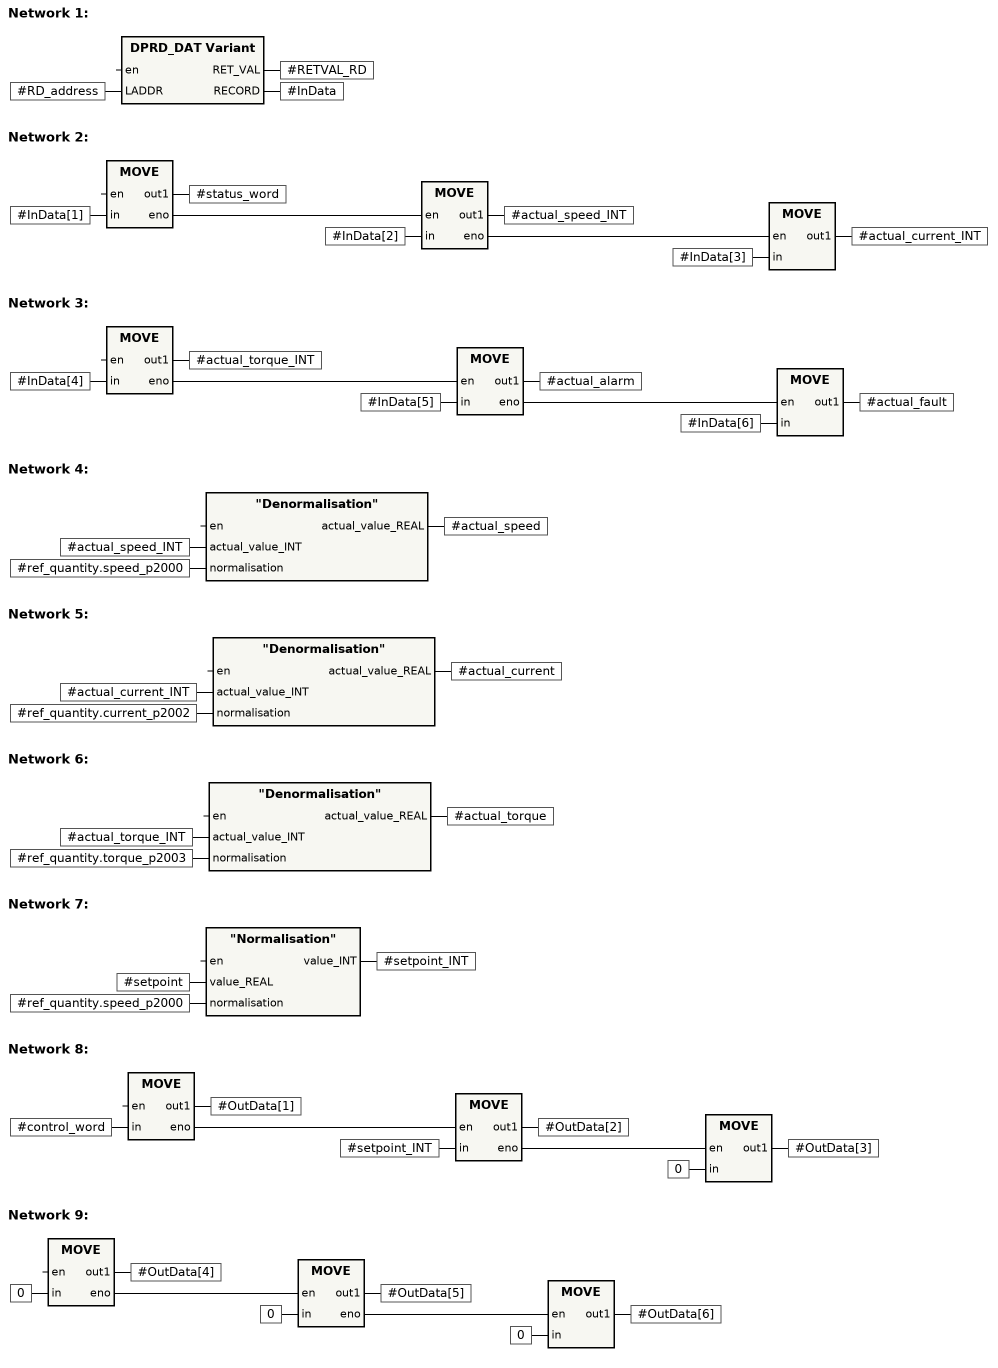
   #RETVAL_RD := DPRD_DAT(LADDR := #RD_address, RECORD => #InData);
END_REGION

REGION Network 2
   // ENO of a box is taken as its EN; it also drops when the box reports an error
   #status_word := #InData[1];
   #actual_speed_INT := #InData[2];
   #actual_current_INT := #InData[3];
END_REGION

REGION Network 3
   // ENO of a box is taken as its EN; it also drops when the box reports an error
   #actual_torque_INT := #InData[4];
   #actual_alarm := #InData[5];
   #actual_fault := #InData[6];
END_REGION

REGION Network 4
   "Denormalisation"(actual_value_INT := #actual_speed_INT,
                     normalisation := #ref_quantity.speed_p2000,
                     actual_value_REAL => #actual_speed);
END_REGION

REGION Network 5
   "Denormalisation"(actual_value_INT := #actual_current_INT,
                     normalisation := #ref_quantity.current_p2002,
                     actual_value_REAL => #actual_current);
END_REGION

REGION Network 6
   "Denormalisation"(actual_value_INT := #actual_torque_INT,
                     normalisation := #ref_quantity.torque_p2003,
                     actual_value_REAL => #actual_torque);
END_REGION

REGION Network 7
   "Normalisation"(value_REAL := #setpoint,
                   normalisation := #ref_quantity.speed_p2000,
                   value_INT => #setpoint_INT);
END_REGION

REGION Network 8
   // ENO of a box is taken as its EN; it also drops when the box reports an error
   #OutData[1] := #control_word;
   #OutData[2] := #setpoint_INT;
   #OutData[3] := 0;
END_REGION

REGION Network 9
   // ENO of a box is taken as its EN; it also drops when the box reports an error
   #OutData[4] := 0;
   #OutData[5] := 0;
   #OutData[6] := 0;
END_REGION

REGION Network 10
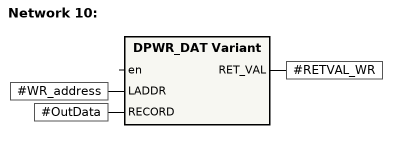
   #RETVAL_WR := DPWR_DAT(LADDR := #WR_address, RECORD := #OutData);
END_REGION
END_FUNCTION_BLOCK

FUNCTION "Denormalisation" : Void   // FC14, FBD
{ S7_Optimized_Access := 'TRUE' }
VERSION : 0.1
// stored: AutoNumber true, IsIECCheckEnabled false, SetENOAutomatically false, UDAEnableTagReadback false
   VAR_INPUT
      actual_value_INT : Int;
      normalisation : Real;
   END_VAR
   VAR_OUTPUT
      actual_value_REAL : Real;
   END_VAR
   VAR_TEMP
      temp_actual_value_DINT : DInt;
      temp_actual_value_REAL : Real;
   END_VAR
BEGIN

REGION Network 1
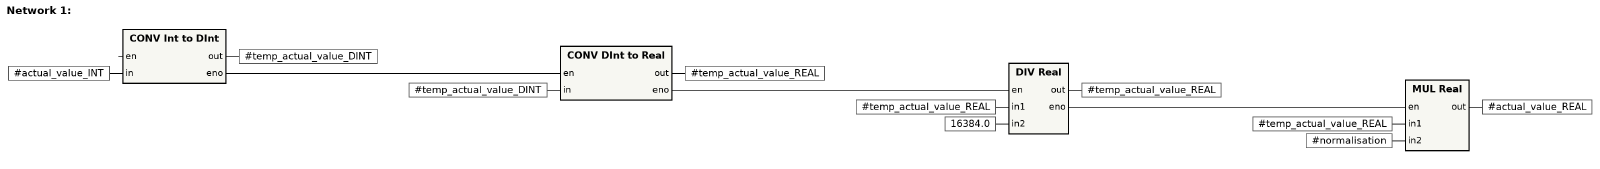
   // ENO of a box is taken as its EN; it also drops when the box reports an error
   #temp_actual_value_DINT := INT_TO_DINT(#actual_value_INT);
   #temp_actual_value_REAL := DINT_TO_REAL(#temp_actual_value_DINT);
   #temp_actual_value_REAL := #temp_actual_value_REAL / 16384.0;
   #actual_value_REAL := #temp_actual_value_REAL * #normalisation;
END_REGION
END_FUNCTION

FUNCTION "Normalisation" : Void   // FC15, FBD
{ S7_Optimized_Access := 'TRUE' }
VERSION : 0.1
// stored: AutoNumber true, IsIECCheckEnabled false, SetENOAutomatically false, UDAEnableTagReadback false
   VAR_INPUT
      value_REAL : Real;
      normalisation : Real;
   END_VAR
   VAR_OUTPUT
      value_INT : Int;
   END_VAR
   VAR_TEMP
      temp_value_DINT : DInt;
      temp_value_REAL : Real;
   END_VAR
BEGIN

REGION Network 1
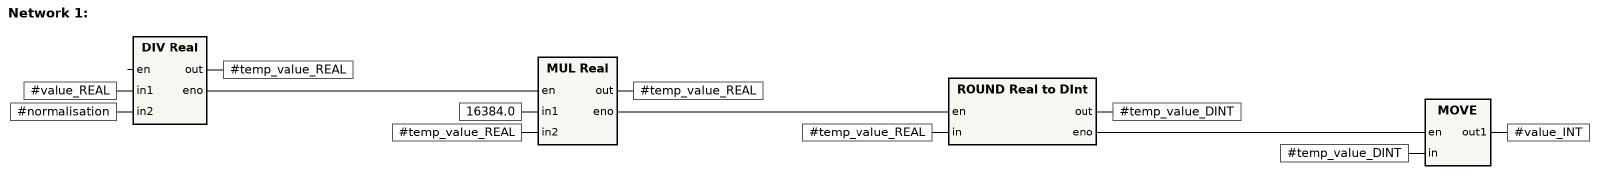
   // ENO of a box is taken as its EN; it also drops when the box reports an error
   #temp_value_REAL := #value_REAL / #normalisation;
   #temp_value_REAL := 16384.0 * #temp_value_REAL;
   #temp_value_DINT := ROUND(#temp_value_REAL);
   #value_INT := #temp_value_DINT;
END_REGION
END_FUNCTION

FUNCTION "FC09_NoPressurePlate" : Void   // FC9, LAD
TITLE = Pressure palte isn't present
{ S7_Optimized_Access := 'FALSE' }
AUTHOR : Robopac
VERSION : 0.0
// stored: AutoNumber false, IsIECCheckEnabled false, SetENOAutomatically false, UDAEnableTagReadback false
BEGIN

REGION Network 1: Pressure plate bits
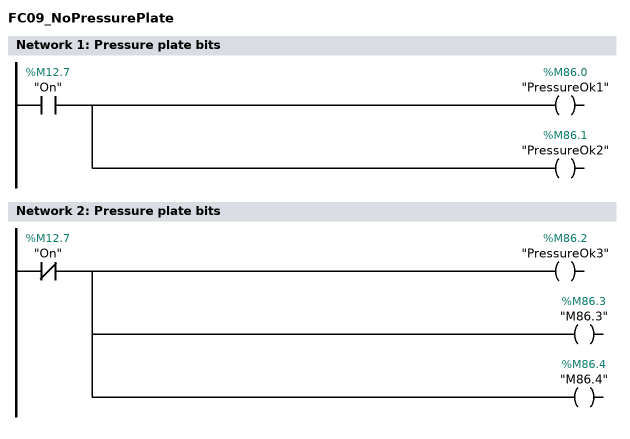
   RUNG wire#powerrail
      Contact( "On" )
      wire#w1
      Coil( "PressureOk1" )
   END_RUNG
   RUNG wire#w1
      Coil( "PressureOk2" )
   END_RUNG
   // the same network as SCL:
   "PressureOk1" := "On";
   "PressureOk2" := "On";
END_REGION

REGION Network 2: Pressure plate bits
   RUNG wire#powerrail
      I_Contact( "On" )
      wire#w1
      Coil( "PressureOk3" )
   END_RUNG
   RUNG wire#w1
      Coil( "M86.3" )
   END_RUNG
   RUNG wire#w1
      Coil( "M86.4" )
   END_RUNG
   // the same network as SCL:
   "PressureOk3" := NOT "On";
   "M86.3" := NOT "On";
   "M86.4" := NOT "On";
END_REGION
END_FUNCTION

FUNCTION "FC11_PressureRectangularPn5W" : Void   // FC11, LAD
{ S7_Optimized_Access := 'FALSE' }
VERSION : 0.1
// stored: AutoNumber false, IsIECCheckEnabled false, SetENOAutomatically false, UDAEnableTagReadback false
BEGIN

REGION Network 1: Timeout for pressure plate upward/downward
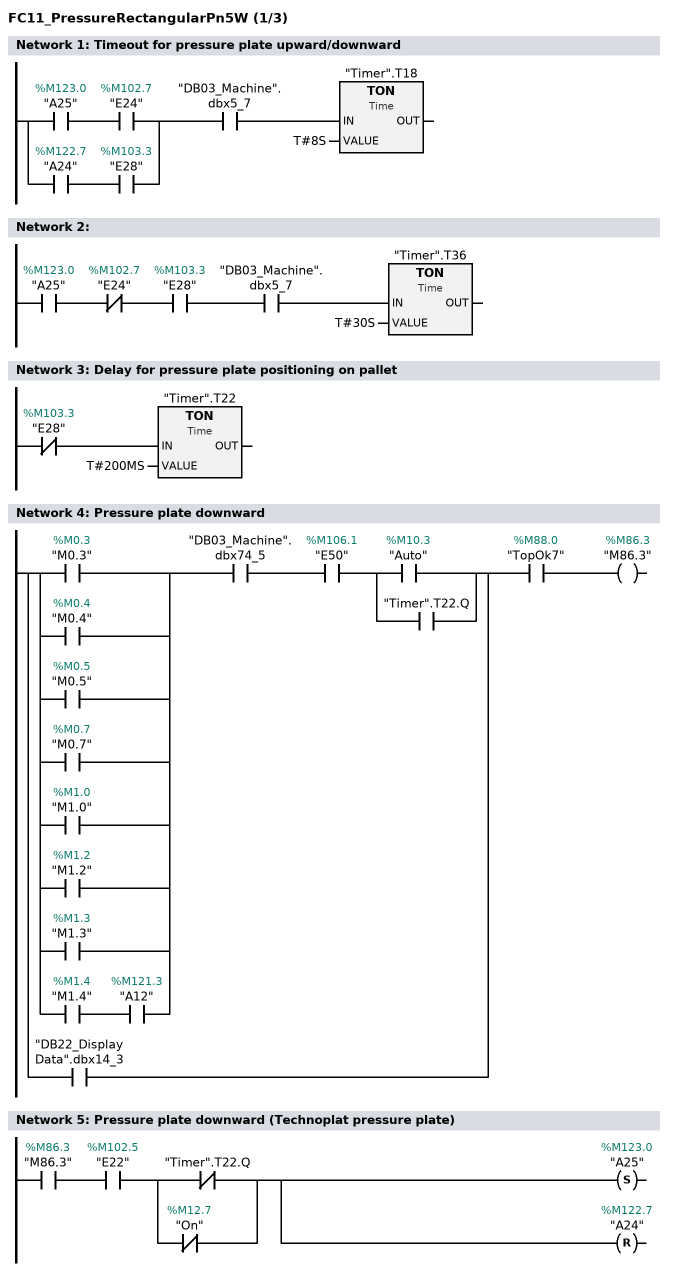
   "Timer".T18.TON(IN := (("A25" AND "E24") OR ("A24" AND "E28")) AND "DB03_Machine".dbx5_7, PT := T#8S);   // TON coil
END_REGION

REGION Network 2
   "Timer".T36.TON(IN := "A25" AND NOT "E24" AND "E28" AND "DB03_Machine".dbx5_7, PT := T#30S);   // TON coil
END_REGION

REGION Network 3: Delay for pressure plate positioning on pallet
   "Timer".T22.TON(IN := NOT "E28", PT := T#200MS);   // TON coil
END_REGION

REGION Network 4: Pressure plate downward
   RUNG wire#powerrail
      Contact( "M0.3" )
      wire#w1
      Contact( "DB03_Machine".dbx74_5 )
      Contact( "E50" )
      wire#w2
      Contact( "Auto" )
      wire#w3
      Contact( "TopOk7" )
      Coil( "M86.3" )
   END_RUNG
   RUNG wire#powerrail
      Contact( "M0.4" )
   END_RUNG wire#w1
   RUNG wire#powerrail
      Contact( "M0.5" )
   END_RUNG wire#w1
   RUNG wire#powerrail
      Contact( "M0.7" )
   END_RUNG wire#w1
   RUNG wire#powerrail
      Contact( "M1.0" )
   END_RUNG wire#w1
   RUNG wire#powerrail
      Contact( "M1.2" )
   END_RUNG wire#w1
   RUNG wire#powerrail
      Contact( "M1.3" )
   END_RUNG wire#w1
   RUNG wire#powerrail
      Contact( "M1.4" )
      Contact( "A12" )
   END_RUNG wire#w1
   RUNG wire#w2
      Contact( "Timer".T22.Q )
   END_RUNG wire#w3
   RUNG wire#powerrail
      Contact( "DB22_DisplayData".dbx14_3 )
   END_RUNG wire#w3
   // the same network as SCL:
   "M86.3" := ((("M0.3" OR "M0.4" OR "M0.5" OR "M0.7" OR "M1.0" OR "M1.2" OR "M1.3" OR ("M1.4" AND "A12")) AND "DB03_Machine".dbx74_5 AND "E50" AND ("Auto" OR "Timer".T22.Q)) OR "DB22_DisplayData".dbx14_3) AND "TopOk7";
END_REGION

REGION Network 5: Pressure plate downward (Technoplat pressure plate)
   RUNG wire#powerrail
      Contact( "M86.3" )
      Contact( "E22" )
      wire#w1
      I_Contact( "Timer".T22.Q )
      wire#w2
      S_Coil( "A25" )
   END_RUNG
   RUNG wire#w1
      I_Contact( "On" )
   END_RUNG wire#w2
   RUNG wire#w2
      R_Coil( "A24" )
   END_RUNG
   // the same network as SCL:
   IF "M86.3" AND "E22" AND (NOT "Timer".T22.Q OR NOT "On") THEN
       "A25" := TRUE;
       "A24" := FALSE;
   END_IF;
END_REGION

REGION Network 6: Pressure plate upward
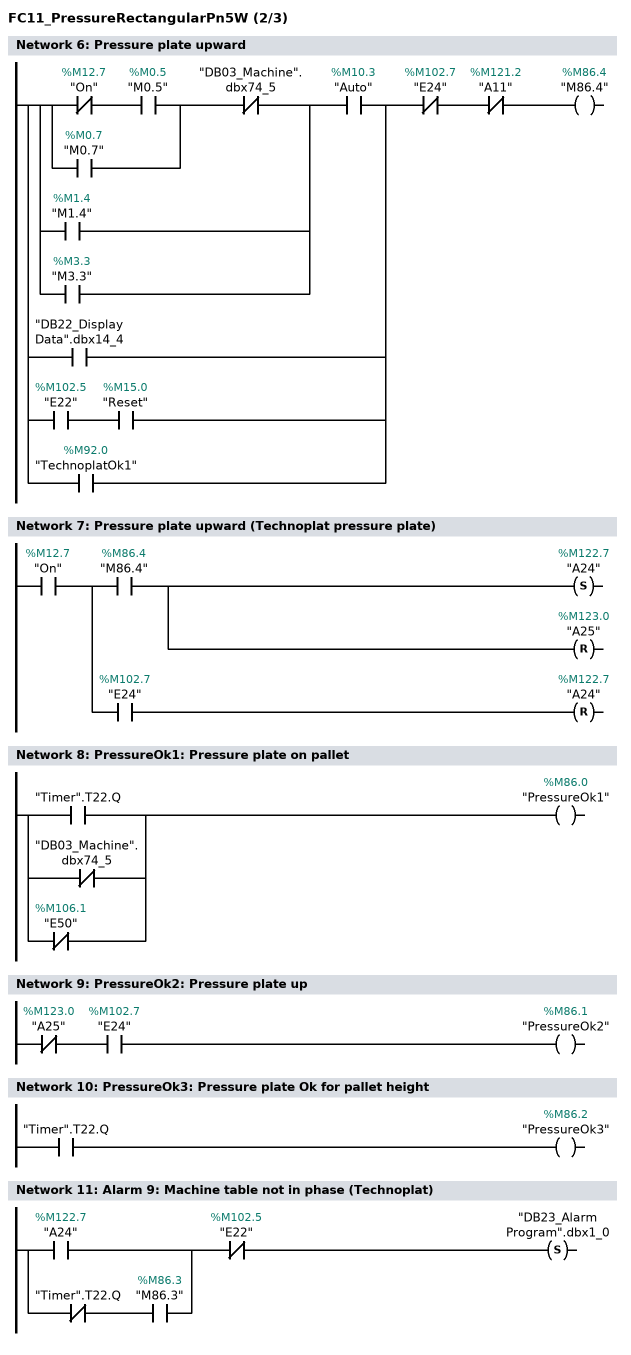
   RUNG wire#powerrail
      I_Contact( "On" )
      Contact( "M0.5" )
      wire#w1
      I_Contact( "DB03_Machine".dbx74_5 )
      wire#w2
      Contact( "Auto" )
      wire#w3
      I_Contact( "E24" )
      I_Contact( "A11" )
      Coil( "M86.4" )
   END_RUNG
   RUNG wire#powerrail
      Contact( "M0.7" )
   END_RUNG wire#w1
   RUNG wire#powerrail
      Contact( "M1.4" )
   END_RUNG wire#w2
   RUNG wire#powerrail
      Contact( "M3.3" )
   END_RUNG wire#w2
   RUNG wire#powerrail
      Contact( "DB22_DisplayData".dbx14_4 )
   END_RUNG wire#w3
   RUNG wire#powerrail
      Contact( "E22" )
      Contact( "Reset" )
   END_RUNG wire#w3
   RUNG wire#powerrail
      Contact( "TechnoplatOk1" )
   END_RUNG wire#w3
   // the same network as SCL:
   "M86.4" := ((((((NOT "On" AND "M0.5") OR "M0.7") AND NOT "DB03_Machine".dbx74_5) OR "M1.4" OR "M3.3") AND "Auto") OR "DB22_DisplayData".dbx14_4 OR ("E22" AND "Reset") OR "TechnoplatOk1") AND NOT "E24" AND NOT "A11";
END_REGION

REGION Network 7: Pressure plate upward (Technoplat pressure plate)
   RUNG wire#powerrail
      Contact( "On" )
      wire#w1
      Contact( "M86.4" )
      wire#w2
      S_Coil( "A24" )
   END_RUNG
   RUNG wire#w2
      R_Coil( "A25" )
   END_RUNG
   RUNG wire#w1
      Contact( "E24" )
      R_Coil( "A24" )
   END_RUNG
   // the same network as SCL:
   IF "On" AND "M86.4" THEN
       "A24" := TRUE;
       "A25" := FALSE;
   END_IF;
   IF "On" AND "E24" THEN "A24" := FALSE; END_IF;
END_REGION

REGION Network 8: PressureOk1: Pressure plate on pallet
   RUNG wire#powerrail
      Contact( "Timer".T22.Q )
      wire#w1
      Coil( "PressureOk1" )
   END_RUNG
   RUNG wire#powerrail
      I_Contact( "DB03_Machine".dbx74_5 )
   END_RUNG wire#w1
   RUNG wire#powerrail
      I_Contact( "E50" )
   END_RUNG wire#w1
   // the same network as SCL:
   "PressureOk1" := "Timer".T22.Q OR NOT "DB03_Machine".dbx74_5 OR NOT "E50";
END_REGION

REGION Network 9: PressureOk2: Pressure plate up
   RUNG wire#powerrail
      I_Contact( "A25" )
      Contact( "E24" )
      Coil( "PressureOk2" )
   END_RUNG
   // the same network as SCL:
   "PressureOk2" := NOT "A25" AND "E24";
END_REGION

REGION Network 10: PressureOk3: Pressure plate Ok for pallet height
   RUNG wire#powerrail
      Contact( "Timer".T22.Q )
      Coil( "PressureOk3" )
   END_RUNG
   // the same network as SCL:
   "PressureOk3" := "Timer".T22.Q;
END_REGION

REGION Network 11: Alarm 9: Machine table not in phase (Technoplat)
   RUNG wire#powerrail
      Contact( "A24" )
      wire#w1
      I_Contact( "E22" )
      S_Coil( "DB23_AlarmProgram".dbx1_0 )
   END_RUNG
   RUNG wire#powerrail
      I_Contact( "Timer".T22.Q )
      Contact( "M86.3" )
   END_RUNG wire#w1
   // the same network as SCL:
   IF ("A24" OR (NOT "Timer".T22.Q AND "M86.3")) AND NOT "E22" THEN
       "DB23_AlarmProgram".dbx1_0 := TRUE;
   END_IF;
END_REGION

REGION Network 12: Alarm 15: Pressure plate not up (Pressure plate)
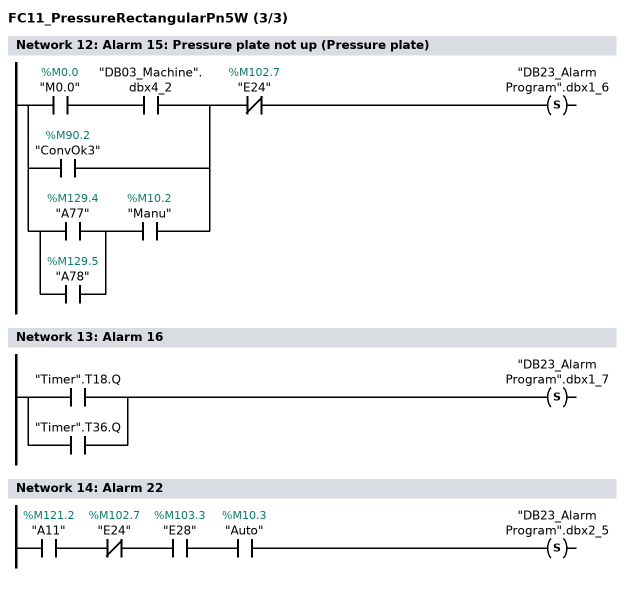
   RUNG wire#powerrail
      Contact( "M0.0" )
      Contact( "DB03_Machine".dbx4_2 )
      wire#w1
      I_Contact( "E24" )
      S_Coil( "DB23_AlarmProgram".dbx1_6 )
   END_RUNG
   RUNG wire#powerrail
      Contact( "ConvOk3" )
   END_RUNG wire#w1
   RUNG wire#powerrail
      Contact( "A77" )
      wire#w2
      Contact( "Manu" )
   END_RUNG wire#w1
   RUNG wire#powerrail
      Contact( "A78" )
   END_RUNG wire#w2
   // the same network as SCL:
   IF (("M0.0" AND "DB03_Machine".dbx4_2) OR "ConvOk3" OR (("A77" OR "A78") AND "Manu")) AND NOT "E24" THEN
       "DB23_AlarmProgram".dbx1_6 := TRUE;
   END_IF;
END_REGION

REGION Network 13: Alarm 16
   RUNG wire#powerrail
      Contact( "Timer".T18.Q )
      wire#w1
      S_Coil( "DB23_AlarmProgram".dbx1_7 )
   END_RUNG
   RUNG wire#powerrail
      Contact( "Timer".T36.Q )
   END_RUNG wire#w1
   // the same network as SCL:
   IF "Timer".T18.Q OR "Timer".T36.Q THEN "DB23_AlarmProgram".dbx1_7 := TRUE; END_IF;
END_REGION

REGION Network 14: Alarm 22
   RUNG wire#powerrail
      Contact( "A11" )
      I_Contact( "E24" )
      Contact( "E28" )
      Contact( "Auto" )
      S_Coil( "DB23_AlarmProgram".dbx2_5 )
   END_RUNG
   // the same network as SCL:
   IF "A11" AND NOT "E24" AND "E28" AND "Auto" THEN "DB23_AlarmProgram".dbx2_5 := TRUE; END_IF;
END_REGION
END_FUNCTION

FUNCTION "FC10_PressureCircularPn5W" : Void   // FC10, LAD
{ S7_Optimized_Access := 'FALSE' }
VERSION : 0.1
// stored: AutoNumber false, IsIECCheckEnabled false, SetENOAutomatically false, UDAEnableTagReadback false
   VAR_TEMP
      PressurePTime : Word;
   END_VAR
   VAR_TEMP   // added for the SCL form of the ladder/FBD networks
      _w1 : Bool;
   END_VAR
BEGIN

REGION Network 1
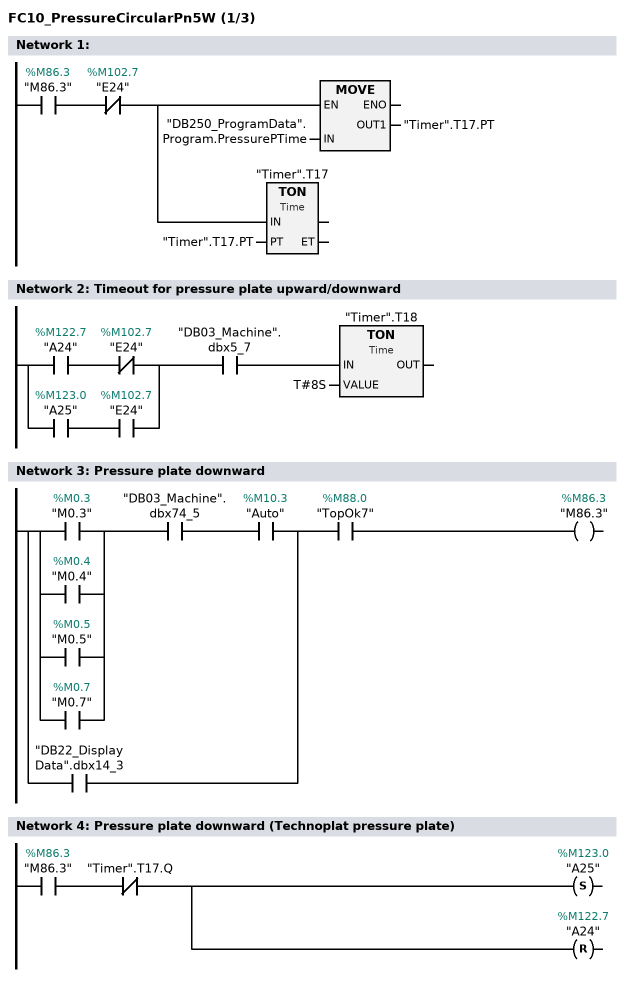
   RUNG wire#powerrail
      Contact( "M86.3" )
      I_Contact( "E24" )
      wire#w1
      { S7_GenerateENO := "TRUE" } Move(in := "DB250_ProgramData".Program.PressurePTime, out1 => "Timer".T17.PT)
   END_RUNG
   RUNG wire#w1
      { S7_Templates := "time_type := Time" } "Timer".T17.TON(pt := "Timer".T17.PT, et =>)
   END_RUNG
   // the same network as SCL:
   #_w1 := "M86.3" AND NOT "E24";
   IF #_w1 THEN "Timer".T17.PT := "DB250_ProgramData".Program.PressurePTime; END_IF;
   "Timer".T17.TON(IN := #_w1, PT := "Timer".T17.PT);
END_REGION

REGION Network 2: Timeout for pressure plate upward/downward
   "Timer".T18.TON(IN := (("A24" AND NOT "E24") OR ("A25" AND "E24")) AND "DB03_Machine".dbx5_7, PT := T#8S);   // TON coil
END_REGION

REGION Network 3: Pressure plate downward
   RUNG wire#powerrail
      Contact( "M0.3" )
      wire#w1
      Contact( "DB03_Machine".dbx74_5 )
      Contact( "Auto" )
      wire#w2
      Contact( "TopOk7" )
      Coil( "M86.3" )
   END_RUNG
   RUNG wire#powerrail
      Contact( "M0.4" )
   END_RUNG wire#w1
   RUNG wire#powerrail
      Contact( "M0.5" )
   END_RUNG wire#w1
   RUNG wire#powerrail
      Contact( "M0.7" )
   END_RUNG wire#w1
   RUNG wire#powerrail
      Contact( "DB22_DisplayData".dbx14_3 )
   END_RUNG wire#w2
   // the same network as SCL:
   "M86.3" := ((("M0.3" OR "M0.4" OR "M0.5" OR "M0.7") AND "DB03_Machine".dbx74_5 AND "Auto") OR "DB22_DisplayData".dbx14_3) AND "TopOk7";
END_REGION

REGION Network 4: Pressure plate downward (Technoplat pressure plate)
   RUNG wire#powerrail
      Contact( "M86.3" )
      I_Contact( "Timer".T17.Q )
      wire#w1
      S_Coil( "A25" )
   END_RUNG
   RUNG wire#w1
      R_Coil( "A24" )
   END_RUNG
   // the same network as SCL:
   IF "M86.3" AND NOT "Timer".T17.Q THEN
       "A25" := TRUE;
       "A24" := FALSE;
   END_IF;
END_REGION

REGION Network 5: Pressure plate upward
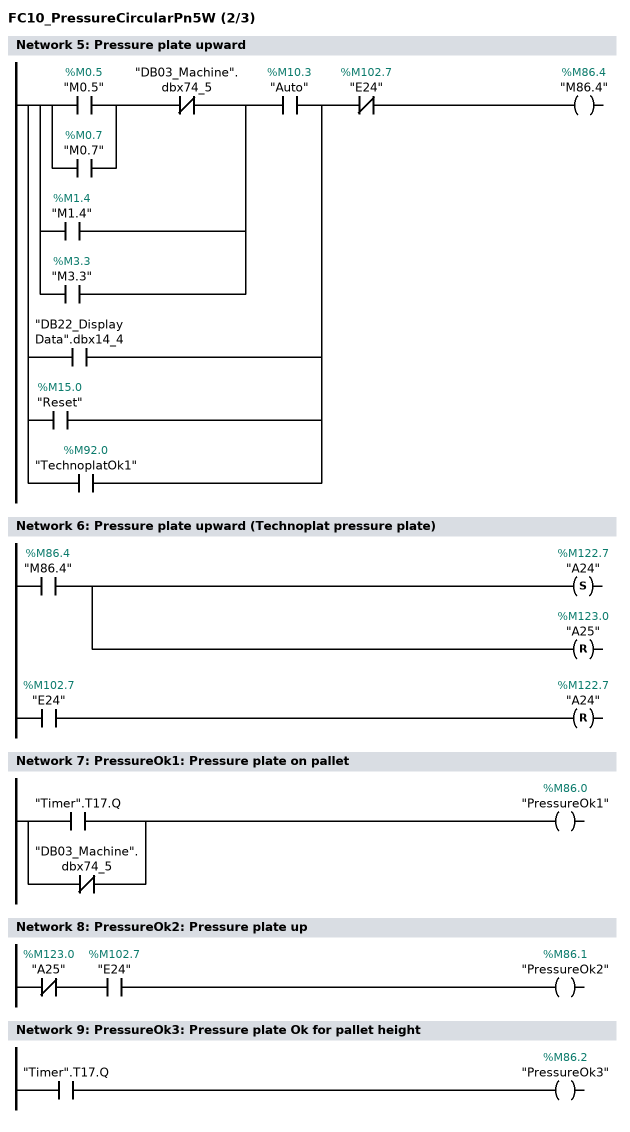
   RUNG wire#powerrail
      Contact( "M0.5" )
      wire#w1
      I_Contact( "DB03_Machine".dbx74_5 )
      wire#w2
      Contact( "Auto" )
      wire#w3
      I_Contact( "E24" )
      Coil( "M86.4" )
   END_RUNG
   RUNG wire#powerrail
      Contact( "M0.7" )
   END_RUNG wire#w1
   RUNG wire#powerrail
      Contact( "M1.4" )
   END_RUNG wire#w2
   RUNG wire#powerrail
      Contact( "M3.3" )
   END_RUNG wire#w2
   RUNG wire#powerrail
      Contact( "DB22_DisplayData".dbx14_4 )
   END_RUNG wire#w3
   RUNG wire#powerrail
      Contact( "Reset" )
   END_RUNG wire#w3
   RUNG wire#powerrail
      Contact( "TechnoplatOk1" )
   END_RUNG wire#w3
   // the same network as SCL:
   "M86.4" := ((((("M0.5" OR "M0.7") AND NOT "DB03_Machine".dbx74_5) OR "M1.4" OR "M3.3") AND "Auto") OR "DB22_DisplayData".dbx14_4 OR "Reset" OR "TechnoplatOk1") AND NOT "E24";
END_REGION

REGION Network 6: Pressure plate upward (Technoplat pressure plate)
   RUNG wire#powerrail
      Contact( "M86.4" )
      wire#w1
      S_Coil( "A24" )
   END_RUNG
   RUNG wire#w1
      R_Coil( "A25" )
   END_RUNG
   RUNG wire#powerrail
      Contact( "E24" )
      R_Coil( "A24" )
   END_RUNG
   // the same network as SCL:
   IF "M86.4" THEN
       "A24" := TRUE;
       "A25" := FALSE;
   END_IF;
   IF "E24" THEN "A24" := FALSE; END_IF;
END_REGION

REGION Network 7: PressureOk1: Pressure plate on pallet
   RUNG wire#powerrail
      Contact( "Timer".T17.Q )
      wire#w1
      Coil( "PressureOk1" )
   END_RUNG
   RUNG wire#powerrail
      I_Contact( "DB03_Machine".dbx74_5 )
   END_RUNG wire#w1
   // the same network as SCL:
   "PressureOk1" := "Timer".T17.Q OR NOT "DB03_Machine".dbx74_5;
END_REGION

REGION Network 8: PressureOk2: Pressure plate up
   RUNG wire#powerrail
      I_Contact( "A25" )
      Contact( "E24" )
      Coil( "PressureOk2" )
   END_RUNG
   // the same network as SCL:
   "PressureOk2" := NOT "A25" AND "E24";
END_REGION

REGION Network 9: PressureOk3: Pressure plate Ok for pallet height
   RUNG wire#powerrail
      Contact( "Timer".T17.Q )
      Coil( "PressureOk3" )
   END_RUNG
   // the same network as SCL:
   "PressureOk3" := "Timer".T17.Q;
END_REGION

REGION Network 10: Alarm 15: Pressure plate not up (Pressure plate)
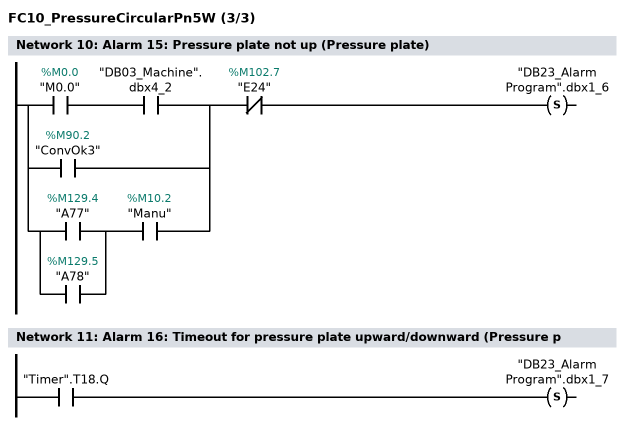
   RUNG wire#powerrail
      Contact( "M0.0" )
      Contact( "DB03_Machine".dbx4_2 )
      wire#w1
      I_Contact( "E24" )
      S_Coil( "DB23_AlarmProgram".dbx1_6 )
   END_RUNG
   RUNG wire#powerrail
      Contact( "ConvOk3" )
   END_RUNG wire#w1
   RUNG wire#powerrail
      Contact( "A77" )
      wire#w2
      Contact( "Manu" )
   END_RUNG wire#w1
   RUNG wire#powerrail
      Contact( "A78" )
   END_RUNG wire#w2
   // the same network as SCL:
   IF (("M0.0" AND "DB03_Machine".dbx4_2) OR "ConvOk3" OR (("A77" OR "A78") AND "Manu")) AND NOT "E24" THEN
       "DB23_AlarmProgram".dbx1_6 := TRUE;
   END_IF;
END_REGION

REGION Network 11: Alarm 16: Timeout for pressure plate upward/downward (Pressure p
   RUNG wire#powerrail
      Contact( "Timer".T18.Q )
      S_Coil( "DB23_AlarmProgram".dbx1_7 )
   END_RUNG
   // the same network as SCL:
   IF "Timer".T18.Q THEN "DB23_AlarmProgram".dbx1_7 := TRUE; END_IF;
END_REGION
END_FUNCTION

FUNCTION "FC12_PressureCircularMono" : Void   // FC12, LAD
{ S7_Optimized_Access := 'FALSE' }
VERSION : 0.1
// stored: AutoNumber false, IsIECCheckEnabled false, SetENOAutomatically false, UDAEnableTagReadback false
   VAR_TEMP
      PressurePTime : Word;
   END_VAR
   VAR_TEMP   // added for the SCL form of the ladder/FBD networks
      _w1 : Bool;
   END_VAR
BEGIN

REGION Network 1
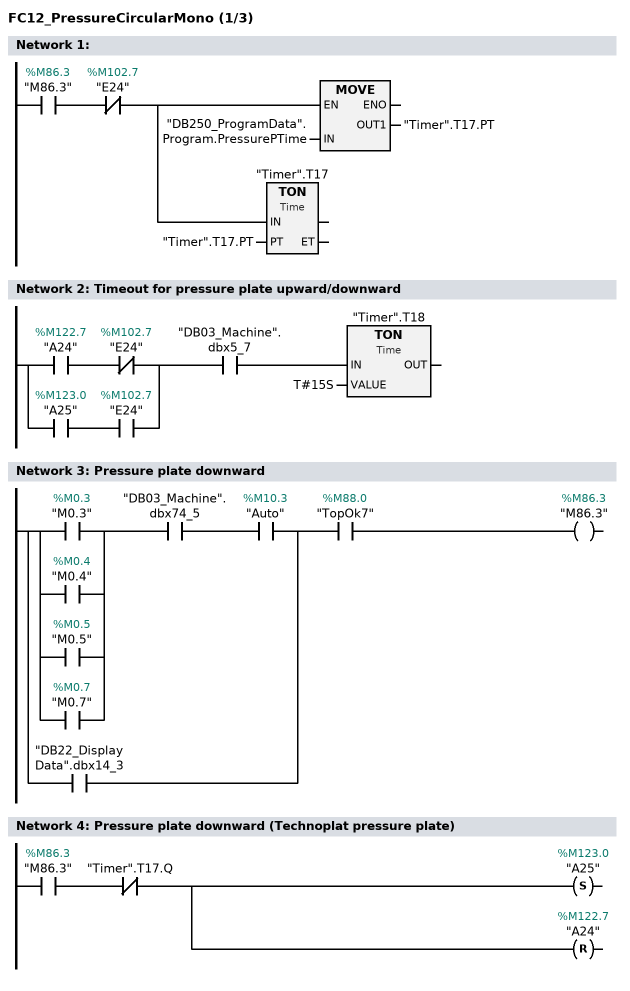
   RUNG wire#powerrail
      Contact( "M86.3" )
      I_Contact( "E24" )
      wire#w1
      { S7_GenerateENO := "TRUE" } Move(in := "DB250_ProgramData".Program.PressurePTime, out1 => "Timer".T17.PT)
   END_RUNG
   RUNG wire#w1
      { S7_Templates := "time_type := Time" } "Timer".T17.TON(pt := "Timer".T17.PT, et =>)
   END_RUNG
   // the same network as SCL:
   #_w1 := "M86.3" AND NOT "E24";
   IF #_w1 THEN "Timer".T17.PT := "DB250_ProgramData".Program.PressurePTime; END_IF;
   "Timer".T17.TON(IN := #_w1, PT := "Timer".T17.PT);
END_REGION

REGION Network 2: Timeout for pressure plate upward/downward
   "Timer".T18.TON(IN := (("A24" AND NOT "E24") OR ("A25" AND "E24")) AND "DB03_Machine".dbx5_7, PT := T#15S);   // TON coil
END_REGION

REGION Network 3: Pressure plate downward
   RUNG wire#powerrail
      Contact( "M0.3" )
      wire#w1
      Contact( "DB03_Machine".dbx74_5 )
      Contact( "Auto" )
      wire#w2
      Contact( "TopOk7" )
      Coil( "M86.3" )
   END_RUNG
   RUNG wire#powerrail
      Contact( "M0.4" )
   END_RUNG wire#w1
   RUNG wire#powerrail
      Contact( "M0.5" )
   END_RUNG wire#w1
   RUNG wire#powerrail
      Contact( "M0.7" )
   END_RUNG wire#w1
   RUNG wire#powerrail
      Contact( "DB22_DisplayData".dbx14_3 )
   END_RUNG wire#w2
   // the same network as SCL:
   "M86.3" := ((("M0.3" OR "M0.4" OR "M0.5" OR "M0.7") AND "DB03_Machine".dbx74_5 AND "Auto") OR "DB22_DisplayData".dbx14_3) AND "TopOk7";
END_REGION

REGION Network 4: Pressure plate downward (Technoplat pressure plate)
   RUNG wire#powerrail
      Contact( "M86.3" )
      I_Contact( "Timer".T17.Q )
      wire#w1
      S_Coil( "A25" )
   END_RUNG
   RUNG wire#w1
      R_Coil( "A24" )
   END_RUNG
   // the same network as SCL:
   IF "M86.3" AND NOT "Timer".T17.Q THEN
       "A25" := TRUE;
       "A24" := FALSE;
   END_IF;
END_REGION

REGION Network 5: Pressure plate upward
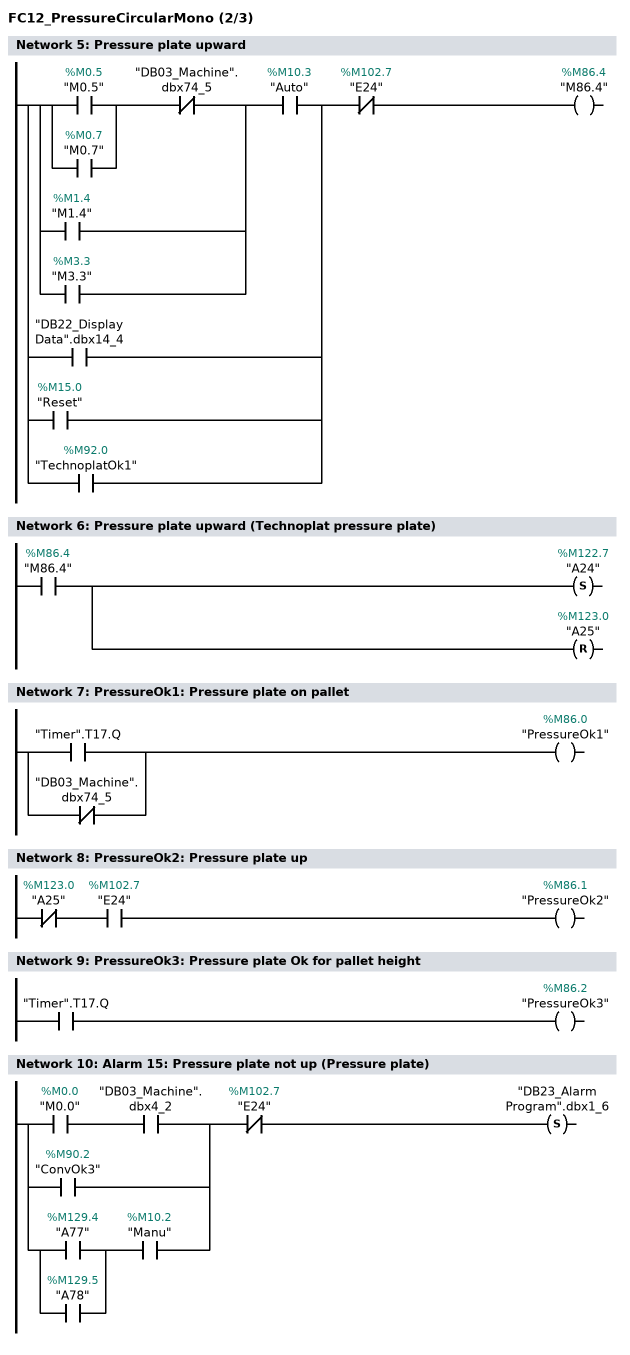
   RUNG wire#powerrail
      Contact( "M0.5" )
      wire#w1
      I_Contact( "DB03_Machine".dbx74_5 )
      wire#w2
      Contact( "Auto" )
      wire#w3
      I_Contact( "E24" )
      Coil( "M86.4" )
   END_RUNG
   RUNG wire#powerrail
      Contact( "M0.7" )
   END_RUNG wire#w1
   RUNG wire#powerrail
      Contact( "M1.4" )
   END_RUNG wire#w2
   RUNG wire#powerrail
      Contact( "M3.3" )
   END_RUNG wire#w2
   RUNG wire#powerrail
      Contact( "DB22_DisplayData".dbx14_4 )
   END_RUNG wire#w3
   RUNG wire#powerrail
      Contact( "Reset" )
   END_RUNG wire#w3
   RUNG wire#powerrail
      Contact( "TechnoplatOk1" )
   END_RUNG wire#w3
   // the same network as SCL:
   "M86.4" := ((((("M0.5" OR "M0.7") AND NOT "DB03_Machine".dbx74_5) OR "M1.4" OR "M3.3") AND "Auto") OR "DB22_DisplayData".dbx14_4 OR "Reset" OR "TechnoplatOk1") AND NOT "E24";
END_REGION

REGION Network 6: Pressure plate upward (Technoplat pressure plate)
   RUNG wire#powerrail
      Contact( "M86.4" )
      wire#w1
      S_Coil( "A24" )
   END_RUNG
   RUNG wire#w1
      R_Coil( "A25" )
   END_RUNG
   // the same network as SCL:
   IF "M86.4" THEN
       "A24" := TRUE;
       "A25" := FALSE;
   END_IF;
END_REGION

REGION Network 7: PressureOk1: Pressure plate on pallet
   RUNG wire#powerrail
      Contact( "Timer".T17.Q )
      wire#w1
      Coil( "PressureOk1" )
   END_RUNG
   RUNG wire#powerrail
      I_Contact( "DB03_Machine".dbx74_5 )
   END_RUNG wire#w1
   // the same network as SCL:
   "PressureOk1" := "Timer".T17.Q OR NOT "DB03_Machine".dbx74_5;
END_REGION

REGION Network 8: PressureOk2: Pressure plate up
   RUNG wire#powerrail
      I_Contact( "A25" )
      Contact( "E24" )
      Coil( "PressureOk2" )
   END_RUNG
   // the same network as SCL:
   "PressureOk2" := NOT "A25" AND "E24";
END_REGION

REGION Network 9: PressureOk3: Pressure plate Ok for pallet height
   RUNG wire#powerrail
      Contact( "Timer".T17.Q )
      Coil( "PressureOk3" )
   END_RUNG
   // the same network as SCL:
   "PressureOk3" := "Timer".T17.Q;
END_REGION

REGION Network 10: Alarm 15: Pressure plate not up (Pressure plate)
   RUNG wire#powerrail
      Contact( "M0.0" )
      Contact( "DB03_Machine".dbx4_2 )
      wire#w1
      I_Contact( "E24" )
      S_Coil( "DB23_AlarmProgram".dbx1_6 )
   END_RUNG
   RUNG wire#powerrail
      Contact( "ConvOk3" )
   END_RUNG wire#w1
   RUNG wire#powerrail
      Contact( "A77" )
      wire#w2
      Contact( "Manu" )
   END_RUNG wire#w1
   RUNG wire#powerrail
      Contact( "A78" )
   END_RUNG wire#w2
   // the same network as SCL:
   IF (("M0.0" AND "DB03_Machine".dbx4_2) OR "ConvOk3" OR (("A77" OR "A78") AND "Manu")) AND NOT "E24" THEN
       "DB23_AlarmProgram".dbx1_6 := TRUE;
   END_IF;
END_REGION

REGION Network 11: Alarm 16: Timeout for pressure plate upward/downward (Pressure p
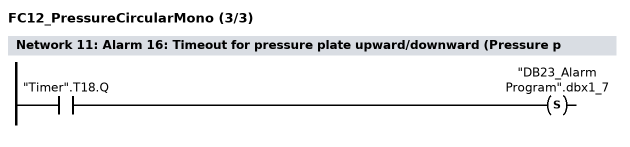
   RUNG wire#powerrail
      Contact( "Timer".T18.Q )
      S_Coil( "DB23_AlarmProgram".dbx1_7 )
   END_RUNG
   // the same network as SCL:
   IF "Timer".T18.Q THEN "DB23_AlarmProgram".dbx1_7 := TRUE; END_IF;
END_REGION
END_FUNCTION

FUNCTION "FC13_TechnoplatClawClamp" : Void   // FC13, LAD
TITLE = Technoplat claw clamp with/without welder unit
{ S7_Optimized_Access := 'FALSE' }
AUTHOR : Robopac
VERSION : 0.0
// stored: AutoNumber false, IsIECCheckEnabled false, SetENOAutomatically false, UDAEnableTagReadback false
   VAR_TEMP   // added for the SCL form of the ladder/FBD networks
      _w1 : Bool;
   END_VAR
BEGIN

REGION Network 1: Welding timer for welder
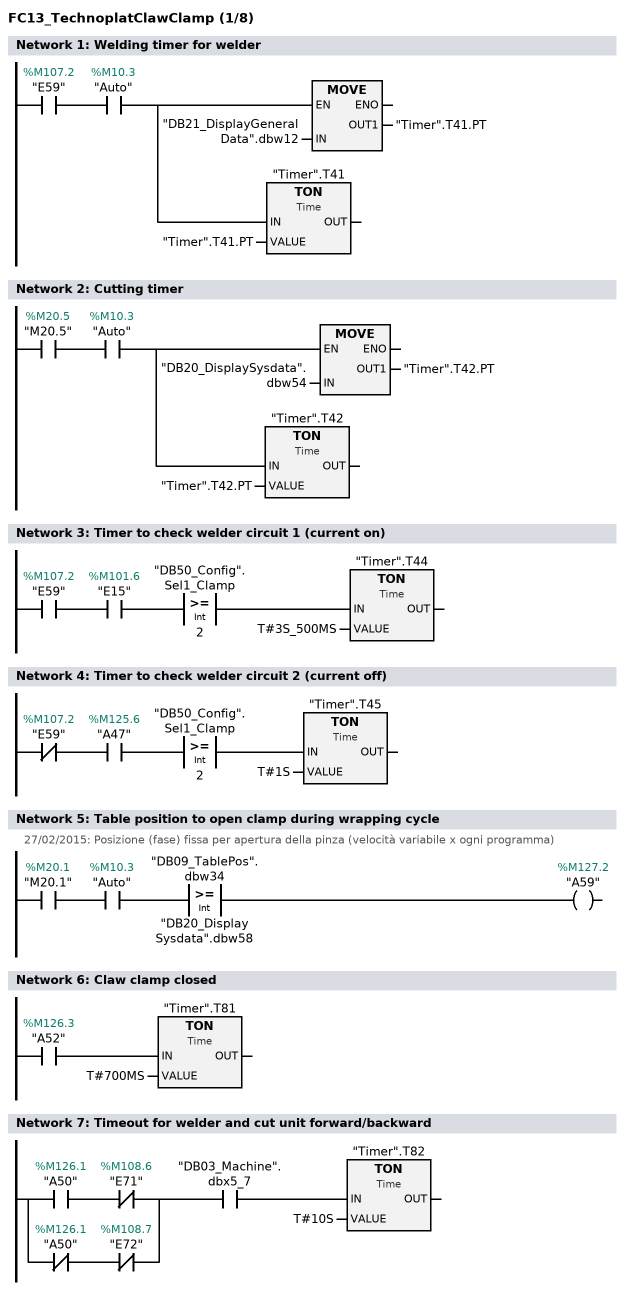
   #_w1 := "E59" AND "Auto";
   IF #_w1 THEN "Timer".T41.PT := "DB21_DisplayGeneralData".dbw12; END_IF;
   "Timer".T41.TON(IN := #_w1, PT := "Timer".T41.PT);   // TON coil
END_REGION

REGION Network 2: Cutting timer
   #_w1 := "M20.5" AND "Auto";
   IF #_w1 THEN "Timer".T42.PT := "DB20_DisplaySysdata".dbw54; END_IF;
   "Timer".T42.TON(IN := #_w1, PT := "Timer".T42.PT);   // TON coil
END_REGION

REGION Network 3: Timer to check welder circuit 1 (current on)
   "Timer".T44.TON(IN := "E59" AND "E15" AND ("DB50_Config".Sel1_Clamp >= 2), PT := T#3S_500MS);   // TON coil
END_REGION

REGION Network 4: Timer to check welder circuit 2 (current off)
   "Timer".T45.TON(IN := NOT "E59" AND "A47" AND ("DB50_Config".Sel1_Clamp >= 2), PT := T#1S);   // TON coil
END_REGION

REGION Network 5: Table position to open clamp during wrapping cycle
   // 27/02/2015: Posizione (fase) fissa per apertura della pinza (velocità variabile x ogni programma)
   RUNG wire#powerrail
      Contact( "M20.1" )
      Contact( "Auto" )
      { S7_Templates := "SrcType := Int" } GE_Contact(in1 := "DB09_TablePos".dbw34, in2 := "DB20_DisplaySysdata".dbw58)
      Coil( "A59" )
   END_RUNG
   // the same network as SCL:
   "A59" := "M20.1" AND "Auto" AND ("DB09_TablePos".dbw34 >= "DB20_DisplaySysdata".dbw58);
END_REGION

REGION Network 6: Claw clamp closed
   "Timer".T81.TON(IN := "A52", PT := T#700MS);   // TON coil
END_REGION

REGION Network 7: Timeout for welder and cut unit forward/backward
   "Timer".T82.TON(IN := (("A50" AND NOT "E71") OR (NOT "A50" AND NOT "E72")) AND "DB03_Machine".dbx5_7, PT := T#10S);   // TON coil
END_REGION

REGION Network 8: Timer for spool carriage movement speed
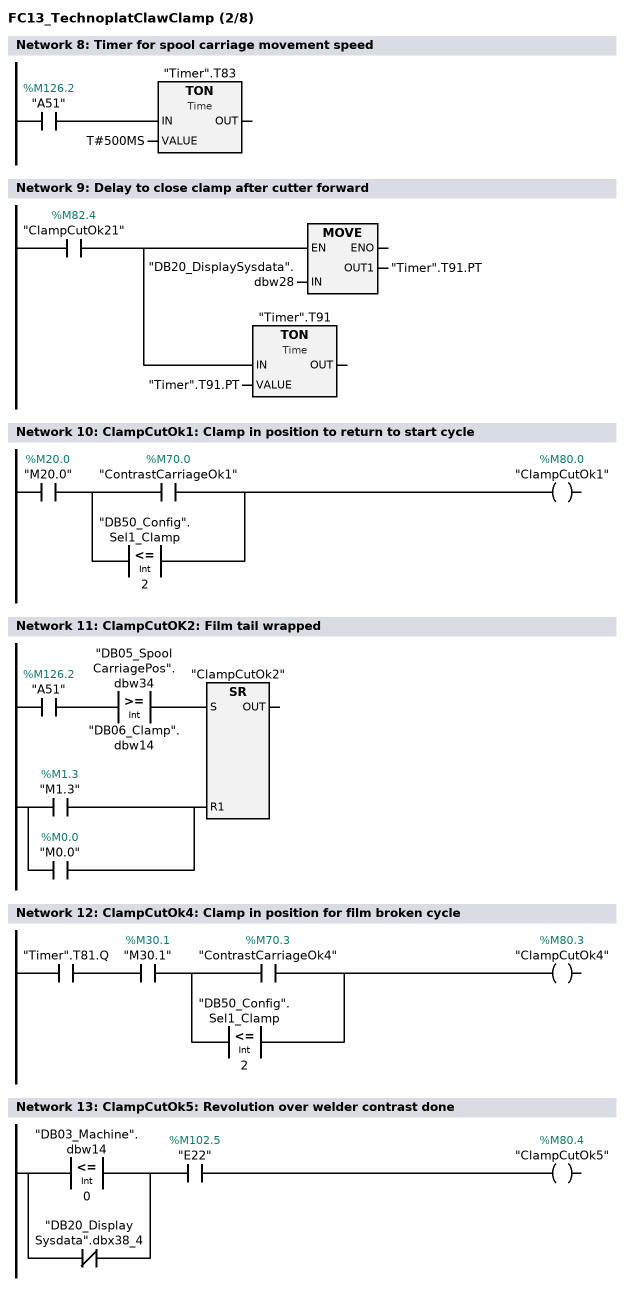
   "Timer".T83.TON(IN := "A51", PT := T#500MS);   // TON coil
END_REGION

REGION Network 9: Delay to close clamp after cutter forward
   IF "ClampCutOk21" THEN "Timer".T91.PT := "DB20_DisplaySysdata".dbw28; END_IF;
   "Timer".T91.TON(IN := "ClampCutOk21", PT := "Timer".T91.PT);   // TON coil
END_REGION

REGION Network 10: ClampCutOk1: Clamp in position to return to start cycle
   RUNG wire#powerrail
      Contact( "M20.0" )
      wire#w1
      Contact( "ContrastCarriageOk1" )
      wire#w2
      Coil( "ClampCutOk1" )
   END_RUNG
   RUNG wire#w1
      { S7_Templates := "SrcType := Int" } LE_Contact(in1 := "DB50_Config".Sel1_Clamp, in2 := 2)
   END_RUNG wire#w2
   // the same network as SCL:
   "ClampCutOk1" := "M20.0" AND ("ContrastCarriageOk1" OR ("DB50_Config".Sel1_Clamp <= 2));
END_REGION

REGION Network 11: ClampCutOK2: Film tail wrapped
   RUNG wire#powerrail
      Contact( "A51" )
      { S7_Templates := "SrcType := Int" } GE_Contact(in1 := "DB05_SpoolCarriagePos".dbw34, in2 := "DB06_Clamp".dbw14)
      S_SR(operand := "ClampCutOk2", r1 := wire#w1)
   END_RUNG
   RUNG wire#powerrail
      Contact( "M1.3" )
   END_RUNG wire#w1
   RUNG wire#powerrail
      Contact( "M0.0" )
   END_RUNG wire#w1
   // the same network as SCL:
   IF "A51" AND ("DB05_SpoolCarriagePos".dbw34 >= "DB06_Clamp".dbw14) THEN
       "ClampCutOk2" := TRUE;   // SR flip-flop
   END_IF;
   IF "M1.3" OR "M0.0" THEN "ClampCutOk2" := FALSE; END_IF;
END_REGION

REGION Network 12: ClampCutOk4: Clamp in position for film broken cycle
   RUNG wire#powerrail
      Contact( "Timer".T81.Q )
      Contact( "M30.1" )
      wire#w1
      Contact( "ContrastCarriageOk4" )
      wire#w2
      Coil( "ClampCutOk4" )
   END_RUNG
   RUNG wire#w1
      { S7_Templates := "SrcType := Int" } LE_Contact(in1 := "DB50_Config".Sel1_Clamp, in2 := 2)
   END_RUNG wire#w2
   // the same network as SCL:
   "ClampCutOk4" := "Timer".T81.Q AND "M30.1" AND ("ContrastCarriageOk4" OR ("DB50_Config".Sel1_Clamp <= 2));
END_REGION

REGION Network 13: ClampCutOk5: Revolution over welder contrast done
   RUNG wire#powerrail
      { S7_Templates := "SrcType := Int" } LE_Contact(in1 := "DB03_Machine".dbw14, in2 := 0)
      wire#w1
      Contact( "E22" )
      Coil( "ClampCutOk5" )
   END_RUNG
   RUNG wire#powerrail
      I_Contact( "DB20_DisplaySysdata".dbx38_4 )
   END_RUNG wire#w1
   // the same network as SCL:
   "ClampCutOk5" := (("DB03_Machine".dbw14 <= 0) OR NOT "DB20_DisplaySysdata".dbx38_4) AND "E22";
END_REGION

REGION Network 14: ClampCutOk6: Clamp and cutter cycle ended
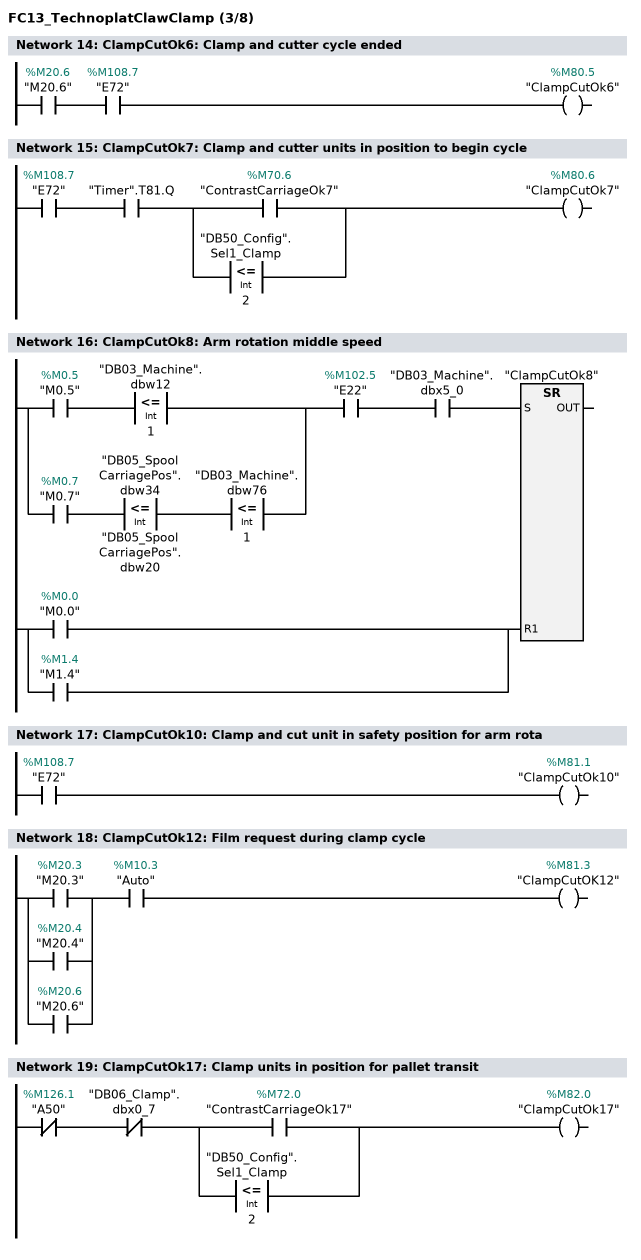
   RUNG wire#powerrail
      Contact( "M20.6" )
      Contact( "E72" )
      Coil( "ClampCutOk6" )
   END_RUNG
   // the same network as SCL:
   "ClampCutOk6" := "M20.6" AND "E72";
END_REGION

REGION Network 15: ClampCutOk7: Clamp and cutter units in position to begin cycle
   RUNG wire#powerrail
      Contact( "E72" )
      Contact( "Timer".T81.Q )
      wire#w1
      Contact( "ContrastCarriageOk7" )
      wire#w2
      Coil( "ClampCutOk7" )
   END_RUNG
   RUNG wire#w1
      { S7_Templates := "SrcType := Int" } LE_Contact(in1 := "DB50_Config".Sel1_Clamp, in2 := 2)
   END_RUNG wire#w2
   // the same network as SCL:
   "ClampCutOk7" := "E72" AND "Timer".T81.Q AND ("ContrastCarriageOk7" OR ("DB50_Config".Sel1_Clamp <= 2));
END_REGION

REGION Network 16: ClampCutOk8: Arm rotation middle speed
   RUNG wire#powerrail
      Contact( "M0.5" )
      { S7_Templates := "SrcType := Int" } LE_Contact(in1 := "DB03_Machine".dbw12, in2 := 1)
      wire#w1
      Contact( "E22" )
      Contact( "DB03_Machine".dbx5_0 )
      S_SR(operand := "ClampCutOk8", r1 := wire#w2)
   END_RUNG
   RUNG wire#powerrail
      Contact( "M0.7" )
      { S7_Templates := "SrcType := Int" } LE_Contact(in1 := "DB05_SpoolCarriagePos".dbw34, in2 := "DB05_SpoolCarriagePos".dbw20)
      { S7_Templates := "SrcType := Int" } LE_Contact(in1 := "DB03_Machine".dbw76, in2 := 1)
   END_RUNG wire#w1
   RUNG wire#powerrail
      Contact( "M0.0" )
   END_RUNG wire#w2
   RUNG wire#powerrail
      Contact( "M1.4" )
   END_RUNG wire#w2
   // the same network as SCL:
   IF (("M0.5" AND ("DB03_Machine".dbw12 <= 1)) OR ("M0.7" AND ("DB05_SpoolCarriagePos".dbw34 <= "DB05_SpoolCarriagePos".dbw20) AND ("DB03_Machine".dbw76 <= 1))) AND "E22" AND "DB03_Machine".dbx5_0 THEN
       "ClampCutOk8" := TRUE;   // SR flip-flop
   END_IF;
   IF "M0.0" OR "M1.4" THEN "ClampCutOk8" := FALSE; END_IF;
END_REGION

REGION Network 17: ClampCutOk10: Clamp and cut unit in safety position for arm rota
   RUNG wire#powerrail
      Contact( "E72" )
      Coil( "ClampCutOk10" )
   END_RUNG
   // the same network as SCL:
   "ClampCutOk10" := "E72";
END_REGION

REGION Network 18: ClampCutOk12: Film request during clamp cycle
   RUNG wire#powerrail
      Contact( "M20.3" )
      wire#w1
      Contact( "Auto" )
      Coil( "ClampCutOK12" )
   END_RUNG
   RUNG wire#powerrail
      Contact( "M20.4" )
   END_RUNG wire#w1
   RUNG wire#powerrail
      Contact( "M20.6" )
   END_RUNG wire#w1
   // the same network as SCL:
   "ClampCutOK12" := ("M20.3" OR "M20.4" OR "M20.6") AND "Auto";
END_REGION

REGION Network 19: ClampCutOk17: Clamp units in position for pallet transit
   RUNG wire#powerrail
      I_Contact( "A50" )
      I_Contact( "DB06_Clamp".dbx0_7 )
      wire#w1
      Contact( "ContrastCarriageOk17" )
      wire#w2
      Coil( "ClampCutOk17" )
   END_RUNG
   RUNG wire#w1
      { S7_Templates := "SrcType := Int" } LE_Contact(in1 := "DB50_Config".Sel1_Clamp, in2 := 2)
   END_RUNG wire#w2
   // the same network as SCL:
   "ClampCutOk17" := NOT "A50" AND NOT "DB06_Clamp".dbx0_7 AND ("ContrastCarriageOk17" OR ("DB50_Config".Sel1_Clamp <= 2));
END_REGION

REGION Network 20: ClampCutOk18: Enable for spool carriage downward at cycle end
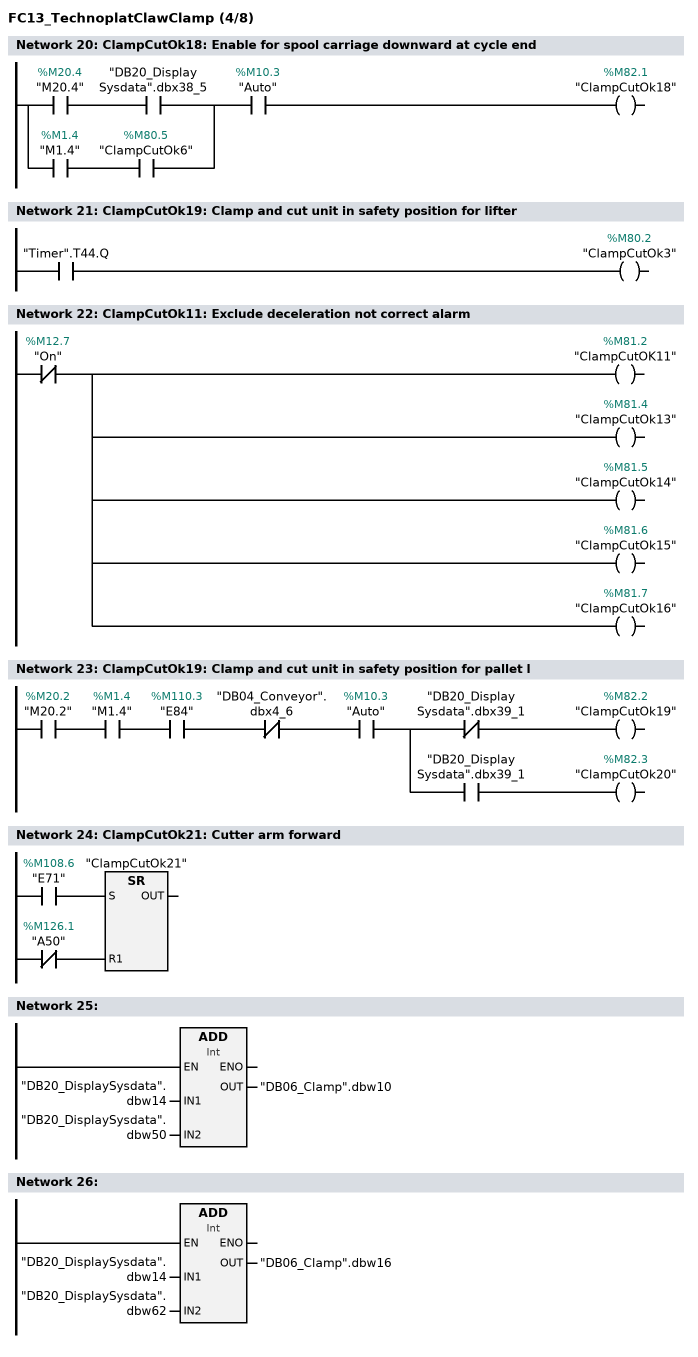
   RUNG wire#powerrail
      Contact( "M20.4" )
      Contact( "DB20_DisplaySysdata".dbx38_5 )
      wire#w1
      Contact( "Auto" )
      Coil( "ClampCutOk18" )
   END_RUNG
   RUNG wire#powerrail
      Contact( "M1.4" )
      Contact( "ClampCutOk6" )
   END_RUNG wire#w1
   // the same network as SCL:
   "ClampCutOk18" := (("M20.4" AND "DB20_DisplaySysdata".dbx38_5) OR ("M1.4" AND "ClampCutOk6")) AND "Auto";
END_REGION

REGION Network 21: ClampCutOk19: Clamp and cut unit in safety position for lifter
   RUNG wire#powerrail
      Contact( "Timer".T44.Q )
      Coil( "ClampCutOk3" )
   END_RUNG
   // the same network as SCL:
   "ClampCutOk3" := "Timer".T44.Q;
END_REGION

REGION Network 22: ClampCutOk11: Exclude deceleration not correct alarm
   RUNG wire#powerrail
      I_Contact( "On" )
      wire#w1
      Coil( "ClampCutOK11" )
   END_RUNG
   RUNG wire#w1
      Coil( "ClampCutOk13" )
   END_RUNG
   RUNG wire#w1
      Coil( "ClampCutOk14" )
   END_RUNG
   RUNG wire#w1
      Coil( "ClampCutOk15" )
   END_RUNG
   RUNG wire#w1
      Coil( "ClampCutOk16" )
   END_RUNG
   // the same network as SCL:
   "ClampCutOK11" := NOT "On";
   "ClampCutOk13" := NOT "On";
   "ClampCutOk14" := NOT "On";
   "ClampCutOk15" := NOT "On";
   "ClampCutOk16" := NOT "On";
END_REGION

REGION Network 23: ClampCutOk19: Clamp and cut unit in safety position for pallet l
   RUNG wire#powerrail
      Contact( "M20.2" )
      Contact( "M1.4" )
      Contact( "E84" )
      I_Contact( "DB04_Conveyor".dbx4_6 )
      Contact( "Auto" )
      wire#w1
      I_Contact( "DB20_DisplaySysdata".dbx39_1 )
      Coil( "ClampCutOk19" )
   END_RUNG
   RUNG wire#w1
      Contact( "DB20_DisplaySysdata".dbx39_1 )
      Coil( "ClampCutOk20" )
   END_RUNG
   // the same network as SCL:
   #_w1 := "M20.2" AND "M1.4" AND "E84" AND NOT "DB04_Conveyor".dbx4_6 AND "Auto";
   "ClampCutOk19" := #_w1 AND NOT "DB20_DisplaySysdata".dbx39_1;
   "ClampCutOk20" := #_w1 AND "DB20_DisplaySysdata".dbx39_1;
END_REGION

REGION Network 24: ClampCutOk21: Cutter arm forward
   RUNG wire#powerrail
      Contact( "E71" )
      S_SR(operand := "ClampCutOk21", r1 := wire#w1)
   END_RUNG
   RUNG wire#powerrail
      I_Contact( "A50" )
   END_RUNG wire#w1
   // the same network as SCL:
   IF "E71" THEN
       "ClampCutOk21" := TRUE;   // SR flip-flop
   END_IF;
   IF NOT "A50" THEN "ClampCutOk21" := FALSE; END_IF;
END_REGION

REGION Network 25
   RUNG wire#powerrail
      { S7_Templates := "SrcType := Int"; S7_GenerateENO := "TRUE" } Add(in1 := "DB20_DisplaySysdata".dbw14, in2 := "DB20_DisplaySysdata".dbw50, out => "DB06_Clamp".dbw10)
   END_RUNG
   // the same network as SCL:
   "DB06_Clamp".dbw10 := "DB20_DisplaySysdata".dbw14 + "DB20_DisplaySysdata".dbw50;
END_REGION

REGION Network 26
   RUNG wire#powerrail
      { S7_Templates := "SrcType := Int"; S7_GenerateENO := "TRUE" } Add(in1 := "DB20_DisplaySysdata".dbw14, in2 := "DB20_DisplaySysdata".dbw62, out => "DB06_Clamp".dbw16)
   END_RUNG
   // the same network as SCL:
   "DB06_Clamp".dbw16 := "DB20_DisplaySysdata".dbw14 + "DB20_DisplaySysdata".dbw62;
END_REGION

REGION Network 27: Number of revolutions to open clamp
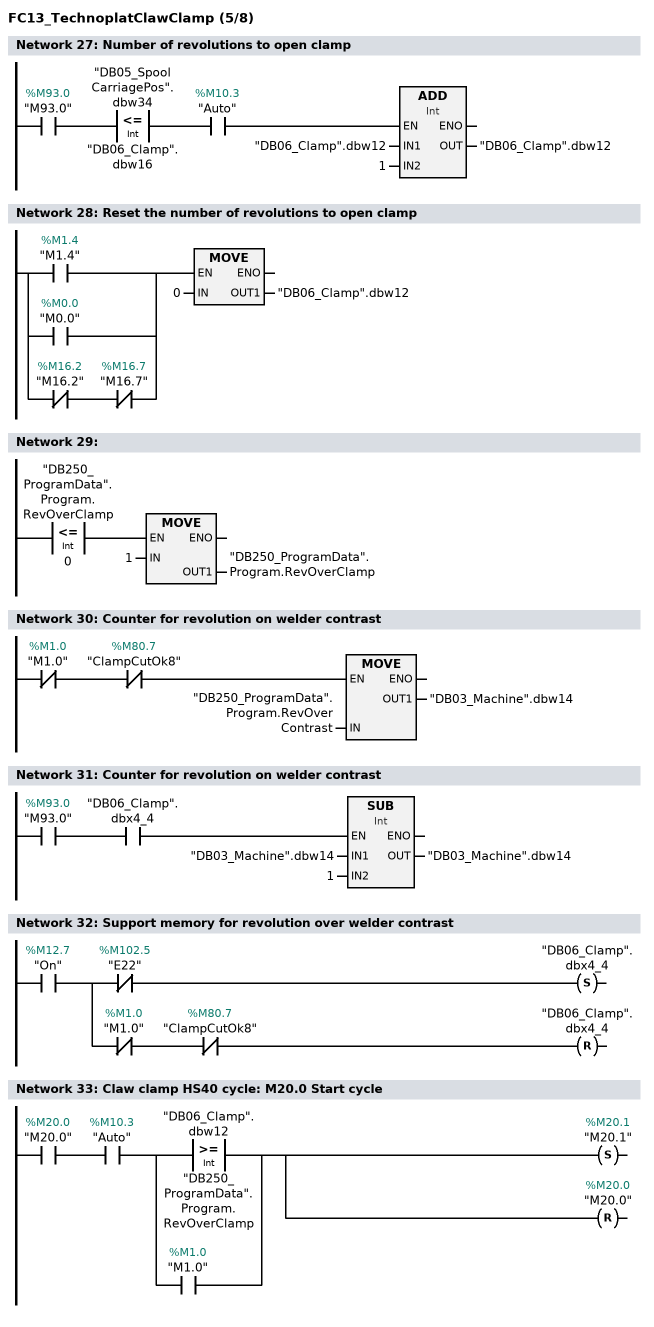
   RUNG wire#powerrail
      Contact( "M93.0" )
      { S7_Templates := "SrcType := Int" } LE_Contact(in1 := "DB05_SpoolCarriagePos".dbw34, in2 := "DB06_Clamp".dbw16)
      Contact( "Auto" )
      { S7_Templates := "SrcType := Int"; S7_GenerateENO := "TRUE" } Add(in1 := "DB06_Clamp".dbw12, in2 := 1, out => "DB06_Clamp".dbw12)
   END_RUNG
   // the same network as SCL:
   IF "M93.0" AND ("DB05_SpoolCarriagePos".dbw34 <= "DB06_Clamp".dbw16) AND "Auto" THEN
       "DB06_Clamp".dbw12 := "DB06_Clamp".dbw12 + 1;
   END_IF;
END_REGION

REGION Network 28: Reset the number of revolutions to open clamp
   RUNG wire#powerrail
      Contact( "M1.4" )
      wire#w1
      { S7_GenerateENO := "TRUE" } Move(in := 0, out1 => "DB06_Clamp".dbw12)
   END_RUNG
   RUNG wire#powerrail
      Contact( "M0.0" )
   END_RUNG wire#w1
   RUNG wire#powerrail
      I_Contact( "M16.2" )
      I_Contact( "M16.7" )
   END_RUNG wire#w1
   // the same network as SCL:
   IF "M1.4" OR "M0.0" OR (NOT "M16.2" AND NOT "M16.7") THEN "DB06_Clamp".dbw12 := 0; END_IF;
END_REGION

REGION Network 29
   RUNG wire#powerrail
      { S7_Templates := "SrcType := Int" } LE_Contact(in1 := "DB250_ProgramData".Program.RevOverClamp, in2 := 0)
      { S7_GenerateENO := "TRUE" } Move(in := 1, out1 => "DB250_ProgramData".Program.RevOverClamp)
   END_RUNG
   // the same network as SCL:
   IF "DB250_ProgramData".Program.RevOverClamp <= 0 THEN
       "DB250_ProgramData".Program.RevOverClamp := 1;
   END_IF;
END_REGION

REGION Network 30: Counter for revolution on welder contrast
   RUNG wire#powerrail
      I_Contact( "M1.0" )
      I_Contact( "ClampCutOk8" )
      { S7_GenerateENO := "TRUE" } Move(in := "DB250_ProgramData".Program.RevOverContrast, out1 => "DB03_Machine".dbw14)
   END_RUNG
   // the same network as SCL:
   IF NOT "M1.0" AND NOT "ClampCutOk8" THEN
       "DB03_Machine".dbw14 := "DB250_ProgramData".Program.RevOverContrast;
   END_IF;
END_REGION

REGION Network 31: Counter for revolution on welder contrast
   RUNG wire#powerrail
      Contact( "M93.0" )
      Contact( "DB06_Clamp".dbx4_4 )
      { S7_Templates := "SrcType := Int"; S7_GenerateENO := "TRUE" } Sub(in1 := "DB03_Machine".dbw14, in2 := 1, out => "DB03_Machine".dbw14)
   END_RUNG
   // the same network as SCL:
   IF "M93.0" AND "DB06_Clamp".dbx4_4 THEN "DB03_Machine".dbw14 := "DB03_Machine".dbw14 - 1; END_IF;
END_REGION

REGION Network 32: Support memory for revolution over welder contrast
   RUNG wire#powerrail
      Contact( "On" )
      wire#w1
      I_Contact( "E22" )
      S_Coil( "DB06_Clamp".dbx4_4 )
   END_RUNG
   RUNG wire#w1
      I_Contact( "M1.0" )
      I_Contact( "ClampCutOk8" )
      R_Coil( "DB06_Clamp".dbx4_4 )
   END_RUNG
   // the same network as SCL:
   IF "On" AND NOT "E22" THEN "DB06_Clamp".dbx4_4 := TRUE; END_IF;
   IF "On" AND NOT "M1.0" AND NOT "ClampCutOk8" THEN "DB06_Clamp".dbx4_4 := FALSE; END_IF;
END_REGION

REGION Network 33: Claw clamp HS40 cycle: M20.0 Start cycle
   RUNG wire#powerrail
      Contact( "M20.0" )
      Contact( "Auto" )
      wire#w1
      { S7_Templates := "SrcType := Int" } GE_Contact(in1 := "DB06_Clamp".dbw12, in2 := "DB250_ProgramData".Program.RevOverClamp)
      wire#w2
      S_Coil( "M20.1" )
   END_RUNG
   RUNG wire#w1
      Contact( "M1.0" )
   END_RUNG wire#w2
   RUNG wire#w2
      R_Coil( "M20.0" )
   END_RUNG
   // the same network as SCL:
   IF "M20.0" AND "Auto" AND (("DB06_Clamp".dbw12 >= "DB250_ProgramData".Program.RevOverClamp) OR "M1.0") THEN
       "M20.1" := TRUE;
       "M20.0" := FALSE;
   END_IF;
END_REGION

REGION Network 34: Claw clamp HS40 cycle: M20.1 Opening clamp
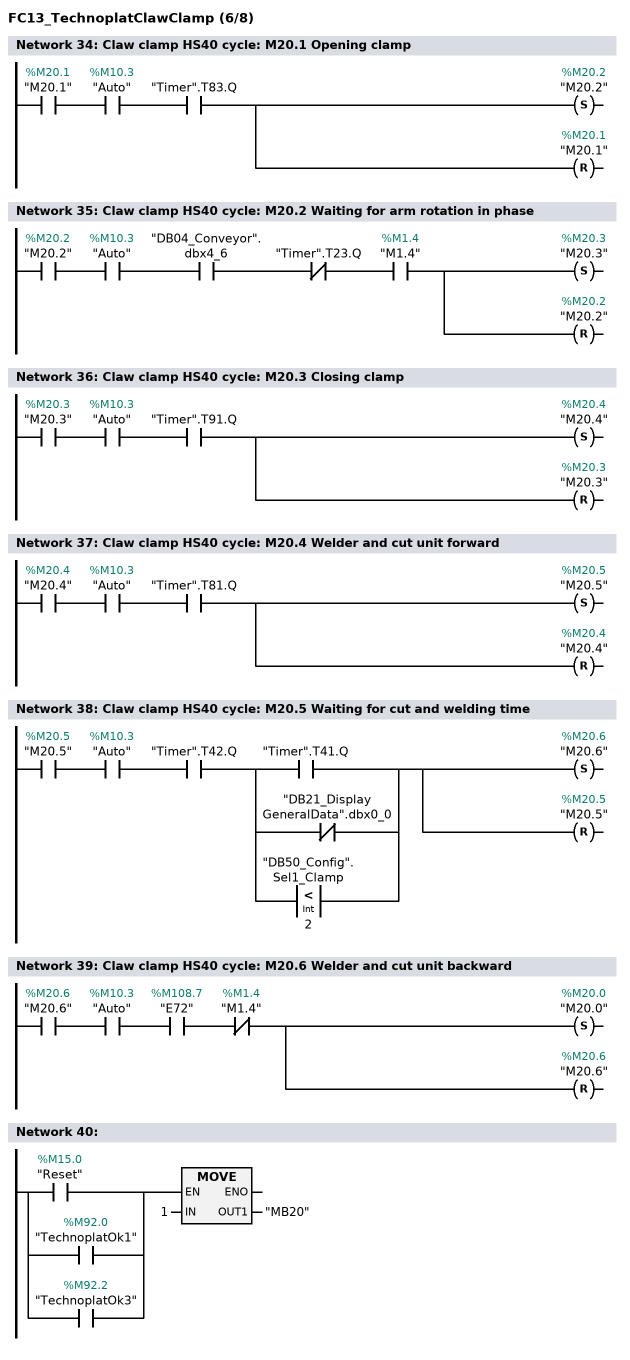
   RUNG wire#powerrail
      Contact( "M20.1" )
      Contact( "Auto" )
      Contact( "Timer".T83.Q )
      wire#w1
      S_Coil( "M20.2" )
   END_RUNG
   RUNG wire#w1
      R_Coil( "M20.1" )
   END_RUNG
   // the same network as SCL:
   IF "M20.1" AND "Auto" AND "Timer".T83.Q THEN
       "M20.2" := TRUE;
       "M20.1" := FALSE;
   END_IF;
END_REGION

REGION Network 35: Claw clamp HS40 cycle: M20.2 Waiting for arm rotation in phase
   RUNG wire#powerrail
      Contact( "M20.2" )
      Contact( "Auto" )
      Contact( "DB04_Conveyor".dbx4_6 )
      I_Contact( "Timer".T23.Q )
      Contact( "M1.4" )
      wire#w1
      S_Coil( "M20.3" )
   END_RUNG
   RUNG wire#w1
      R_Coil( "M20.2" )
   END_RUNG
   // the same network as SCL:
   IF "M20.2" AND "Auto" AND "DB04_Conveyor".dbx4_6 AND NOT "Timer".T23.Q AND "M1.4" THEN
       "M20.3" := TRUE;
       "M20.2" := FALSE;
   END_IF;
END_REGION

REGION Network 36: Claw clamp HS40 cycle: M20.3 Closing clamp
   RUNG wire#powerrail
      Contact( "M20.3" )
      Contact( "Auto" )
      Contact( "Timer".T91.Q )
      wire#w1
      S_Coil( "M20.4" )
   END_RUNG
   RUNG wire#w1
      R_Coil( "M20.3" )
   END_RUNG
   // the same network as SCL:
   IF "M20.3" AND "Auto" AND "Timer".T91.Q THEN
       "M20.4" := TRUE;
       "M20.3" := FALSE;
   END_IF;
END_REGION

REGION Network 37: Claw clamp HS40 cycle: M20.4 Welder and cut unit forward
   RUNG wire#powerrail
      Contact( "M20.4" )
      Contact( "Auto" )
      Contact( "Timer".T81.Q )
      wire#w1
      S_Coil( "M20.5" )
   END_RUNG
   RUNG wire#w1
      R_Coil( "M20.4" )
   END_RUNG
   // the same network as SCL:
   IF "M20.4" AND "Auto" AND "Timer".T81.Q THEN
       "M20.5" := TRUE;
       "M20.4" := FALSE;
   END_IF;
END_REGION

REGION Network 38: Claw clamp HS40 cycle: M20.5 Waiting for cut and welding time
   RUNG wire#powerrail
      Contact( "M20.5" )
      Contact( "Auto" )
      Contact( "Timer".T42.Q )
      wire#w1
      Contact( "Timer".T41.Q )
      wire#w2
      S_Coil( "M20.6" )
   END_RUNG
   RUNG wire#w1
      I_Contact( "DB21_DisplayGeneralData".dbx0_0 )
   END_RUNG wire#w2
   RUNG wire#w1
      { S7_Templates := "SrcType := Int" } LT_Contact(in1 := "DB50_Config".Sel1_Clamp, in2 := 2)
   END_RUNG wire#w2
   RUNG wire#w2
      R_Coil( "M20.5" )
   END_RUNG
   // the same network as SCL:
   IF "M20.5" AND "Auto" AND "Timer".T42.Q AND ("Timer".T41.Q OR NOT "DB21_DisplayGeneralData".dbx0_0 OR ("DB50_Config".Sel1_Clamp < 2)) THEN
       "M20.6" := TRUE;
       "M20.5" := FALSE;
   END_IF;
END_REGION

REGION Network 39: Claw clamp HS40 cycle: M20.6 Welder and cut unit backward
   RUNG wire#powerrail
      Contact( "M20.6" )
      Contact( "Auto" )
      Contact( "E72" )
      I_Contact( "M1.4" )
      wire#w1
      S_Coil( "M20.0" )
   END_RUNG
   RUNG wire#w1
      R_Coil( "M20.6" )
   END_RUNG
   // the same network as SCL:
   IF "M20.6" AND "Auto" AND "E72" AND NOT "M1.4" THEN
       "M20.0" := TRUE;
       "M20.6" := FALSE;
   END_IF;
END_REGION

REGION Network 40
   RUNG wire#powerrail
      Contact( "Reset" )
      wire#w1
      { S7_GenerateENO := "TRUE" } Move(in := 1, out1 => "MB20")
   END_RUNG
   RUNG wire#powerrail
      Contact( "TechnoplatOk1" )
   END_RUNG wire#w1
   RUNG wire#powerrail
      Contact( "TechnoplatOk3" )
   END_RUNG wire#w1
   // the same network as SCL:
   IF "Reset" OR "TechnoplatOk1" OR "TechnoplatOk3" THEN "MB20" := 1; END_IF;
END_REGION

REGION Network 41: Film clamp opening (Claw clamp)
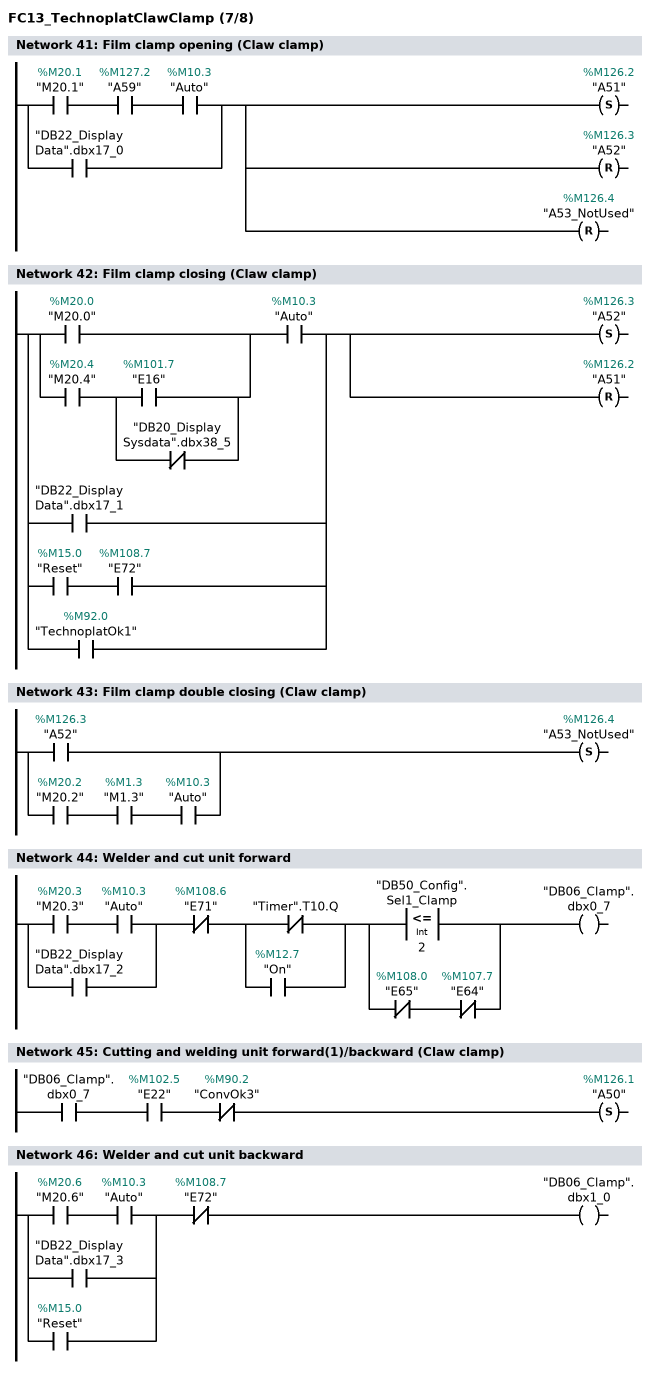
   RUNG wire#powerrail
      Contact( "M20.1" )
      Contact( "A59" )
      Contact( "Auto" )
      wire#w1
      S_Coil( "A51" )
   END_RUNG
   RUNG wire#powerrail
      Contact( "DB22_DisplayData".dbx17_0 )
   END_RUNG wire#w1
   RUNG wire#w1
      R_Coil( "A52" )
   END_RUNG
   RUNG wire#w1
      R_Coil( "A53_NotUsed" )
   END_RUNG
   // the same network as SCL:
   IF ("M20.1" AND "A59" AND "Auto") OR "DB22_DisplayData".dbx17_0 THEN
       "A51" := TRUE;
       "A52" := FALSE;
       "A53_NotUsed" := FALSE;
   END_IF;
END_REGION

REGION Network 42: Film clamp closing (Claw clamp)
   RUNG wire#powerrail
      Contact( "M20.0" )
      wire#w1
      Contact( "Auto" )
      wire#w3
      S_Coil( "A52" )
   END_RUNG
   RUNG wire#powerrail
      Contact( "M20.4" )
      wire#w2
      Contact( "E16" )
   END_RUNG wire#w1
   RUNG wire#w2
      I_Contact( "DB20_DisplaySysdata".dbx38_5 )
   END_RUNG wire#w1
   RUNG wire#powerrail
      Contact( "DB22_DisplayData".dbx17_1 )
   END_RUNG wire#w3
   RUNG wire#powerrail
      Contact( "Reset" )
      Contact( "E72" )
   END_RUNG wire#w3
   RUNG wire#powerrail
      Contact( "TechnoplatOk1" )
   END_RUNG wire#w3
   RUNG wire#w3
      R_Coil( "A51" )
   END_RUNG
   // the same network as SCL:
   IF (("M20.0" OR ("M20.4" AND ("E16" OR NOT "DB20_DisplaySysdata".dbx38_5))) AND "Auto") OR "DB22_DisplayData".dbx17_1 OR ("Reset" AND "E72") OR "TechnoplatOk1" THEN
       "A52" := TRUE;
       "A51" := FALSE;
   END_IF;
END_REGION

REGION Network 43: Film clamp double closing (Claw clamp)
   RUNG wire#powerrail
      Contact( "A52" )
      wire#w1
      S_Coil( "A53_NotUsed" )
   END_RUNG
   RUNG wire#powerrail
      Contact( "M20.2" )
      Contact( "M1.3" )
      Contact( "Auto" )
   END_RUNG wire#w1
   // the same network as SCL:
   IF "A52" OR ("M20.2" AND "M1.3" AND "Auto") THEN "A53_NotUsed" := TRUE; END_IF;
END_REGION

REGION Network 44: Welder and cut unit forward
   RUNG wire#powerrail
      Contact( "M20.3" )
      Contact( "Auto" )
      wire#w1
      I_Contact( "E71" )
      wire#w2
      I_Contact( "Timer".T10.Q )
      wire#w3
      { S7_Templates := "SrcType := Int" } LE_Contact(in1 := "DB50_Config".Sel1_Clamp, in2 := 2)
      wire#w4
      Coil( "DB06_Clamp".dbx0_7 )
   END_RUNG
   RUNG wire#powerrail
      Contact( "DB22_DisplayData".dbx17_2 )
   END_RUNG wire#w1
   RUNG wire#w2
      Contact( "On" )
   END_RUNG wire#w3
   RUNG wire#w3
      I_Contact( "E65" )
      I_Contact( "E64" )
   END_RUNG wire#w4
   // the same network as SCL:
   "DB06_Clamp".dbx0_7 := (("M20.3" AND "Auto") OR "DB22_DisplayData".dbx17_2) AND NOT "E71" AND (NOT "Timer".T10.Q OR "On") AND (("DB50_Config".Sel1_Clamp <= 2) OR (NOT "E65" AND NOT "E64"));
END_REGION

REGION Network 45: Cutting and welding unit forward(1)/backward (Claw clamp)
   RUNG wire#powerrail
      Contact( "DB06_Clamp".dbx0_7 )
      Contact( "E22" )
      I_Contact( "ConvOk3" )
      S_Coil( "A50" )
   END_RUNG
   // the same network as SCL:
   IF "DB06_Clamp".dbx0_7 AND "E22" AND NOT "ConvOk3" THEN "A50" := TRUE; END_IF;
END_REGION

REGION Network 46: Welder and cut unit backward
   RUNG wire#powerrail
      Contact( "M20.6" )
      Contact( "Auto" )
      wire#w1
      I_Contact( "E72" )
      Coil( "DB06_Clamp".dbx1_0 )
   END_RUNG
   RUNG wire#powerrail
      Contact( "DB22_DisplayData".dbx17_3 )
   END_RUNG wire#w1
   RUNG wire#powerrail
      Contact( "Reset" )
   END_RUNG wire#w1
   // the same network as SCL:
   "DB06_Clamp".dbx1_0 := (("M20.6" AND "Auto") OR "DB22_DisplayData".dbx17_3 OR "Reset") AND NOT "E72";
END_REGION

REGION Network 47: Cutting and welding unit forward(1)/backward (Claw clamp)
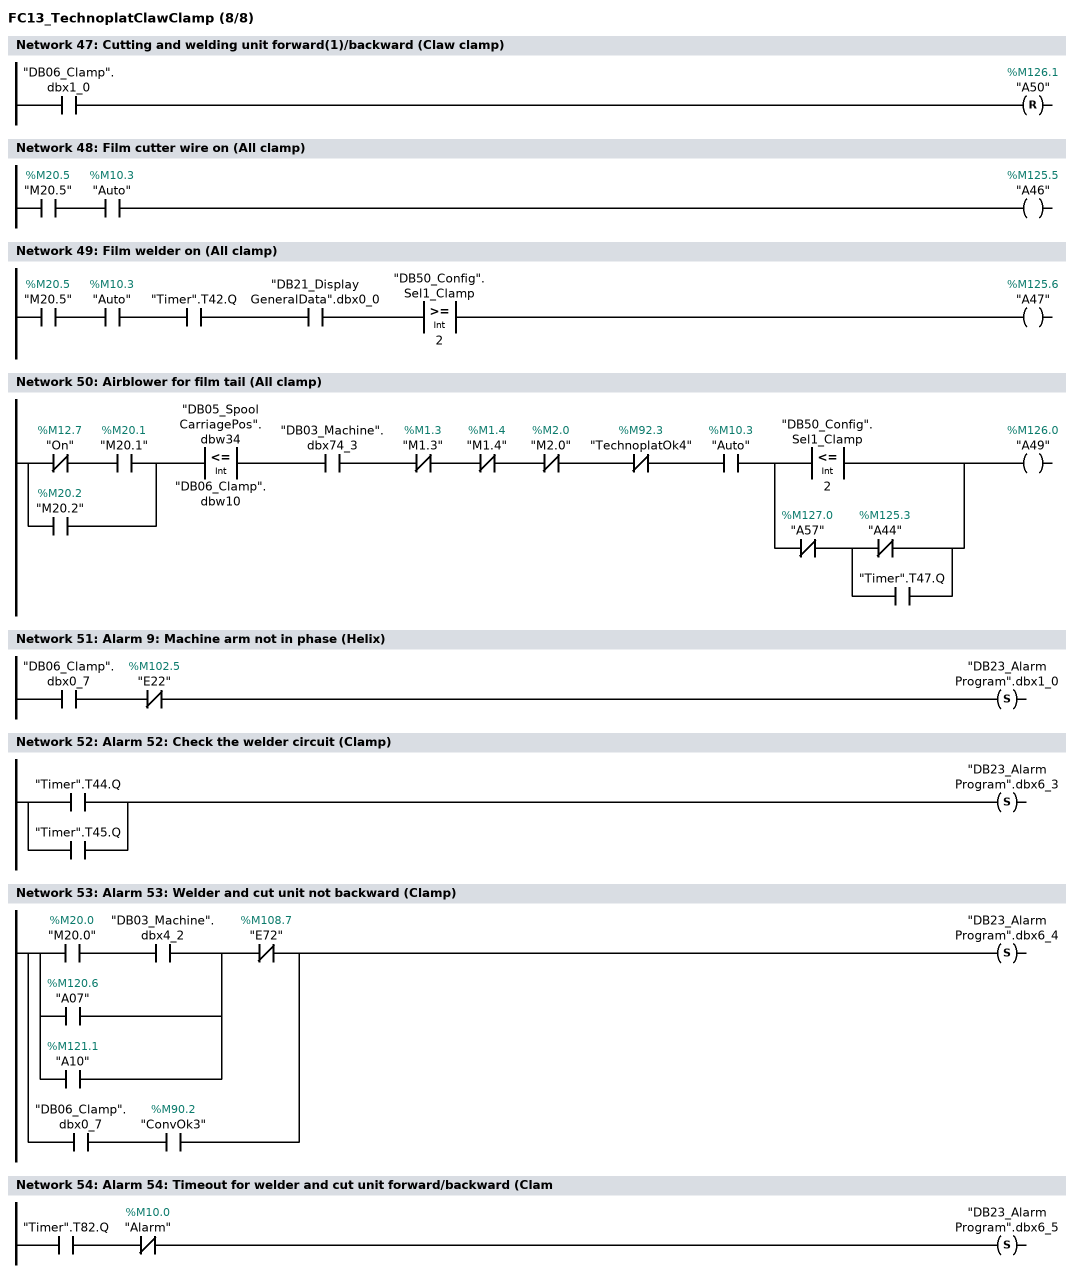
   RUNG wire#powerrail
      Contact( "DB06_Clamp".dbx1_0 )
      R_Coil( "A50" )
   END_RUNG
   // the same network as SCL:
   IF "DB06_Clamp".dbx1_0 THEN "A50" := FALSE; END_IF;
END_REGION

REGION Network 48: Film cutter wire on (All clamp)
   RUNG wire#powerrail
      Contact( "M20.5" )
      Contact( "Auto" )
      Coil( "A46" )
   END_RUNG
   // the same network as SCL:
   "A46" := "M20.5" AND "Auto";
END_REGION

REGION Network 49: Film welder on (All clamp)
   RUNG wire#powerrail
      Contact( "M20.5" )
      Contact( "Auto" )
      Contact( "Timer".T42.Q )
      Contact( "DB21_DisplayGeneralData".dbx0_0 )
      { S7_Templates := "SrcType := Int" } GE_Contact(in1 := "DB50_Config".Sel1_Clamp, in2 := 2)
      Coil( "A47" )
   END_RUNG
   // the same network as SCL:
   "A47" := "M20.5" AND "Auto" AND "Timer".T42.Q AND "DB21_DisplayGeneralData".dbx0_0 AND ("DB50_Config".Sel1_Clamp >= 2);
END_REGION

REGION Network 50: Airblower for film tail (All clamp)
   RUNG wire#powerrail
      I_Contact( "On" )
      Contact( "M20.1" )
      wire#w1
      { S7_Templates := "SrcType := Int" } LE_Contact(in1 := "DB05_SpoolCarriagePos".dbw34, in2 := "DB06_Clamp".dbw10)
      Contact( "DB03_Machine".dbx74_3 )
      I_Contact( "M1.3" )
      I_Contact( "M1.4" )
      I_Contact( "M2.0" )
      I_Contact( "TechnoplatOk4" )
      Contact( "Auto" )
      wire#w2
      { S7_Templates := "SrcType := Int" } LE_Contact(in1 := "DB50_Config".Sel1_Clamp, in2 := 2)
      wire#w3
      Coil( "A49" )
   END_RUNG
   RUNG wire#powerrail
      Contact( "M20.2" )
   END_RUNG wire#w1
   RUNG wire#w2
      I_Contact( "A57" )
      wire#w4
      I_Contact( "A44" )
   END_RUNG wire#w3
   RUNG wire#w4
      Contact( "Timer".T47.Q )
   END_RUNG wire#w3
   // the same network as SCL:
   "A49" := ((NOT "On" AND "M20.1") OR "M20.2") AND ("DB05_SpoolCarriagePos".dbw34 <= "DB06_Clamp".dbw10) AND "DB03_Machine".dbx74_3 AND NOT "M1.3" AND NOT "M1.4" AND NOT "M2.0" AND NOT "TechnoplatOk4" AND "Auto" AND (("DB50_Config".Sel1_Clamp <= 2) OR (NOT "A57" AND (NOT "A44" OR "Timer".T47.Q)));
END_REGION

REGION Network 51: Alarm 9: Machine arm not in phase (Helix)
   RUNG wire#powerrail
      Contact( "DB06_Clamp".dbx0_7 )
      I_Contact( "E22" )
      S_Coil( "DB23_AlarmProgram".dbx1_0 )
   END_RUNG
   // the same network as SCL:
   IF "DB06_Clamp".dbx0_7 AND NOT "E22" THEN "DB23_AlarmProgram".dbx1_0 := TRUE; END_IF;
END_REGION

REGION Network 52: Alarm 52: Check the welder circuit (Clamp)
   RUNG wire#powerrail
      Contact( "Timer".T44.Q )
      wire#w1
      S_Coil( "DB23_AlarmProgram".dbx6_3 )
   END_RUNG
   RUNG wire#powerrail
      Contact( "Timer".T45.Q )
   END_RUNG wire#w1
   // the same network as SCL:
   IF "Timer".T44.Q OR "Timer".T45.Q THEN "DB23_AlarmProgram".dbx6_3 := TRUE; END_IF;
END_REGION

REGION Network 53: Alarm 53: Welder and cut unit not backward (Clamp)
   RUNG wire#powerrail
      Contact( "M20.0" )
      Contact( "DB03_Machine".dbx4_2 )
      wire#w1
      I_Contact( "E72" )
      wire#w2
      S_Coil( "DB23_AlarmProgram".dbx6_4 )
   END_RUNG
   RUNG wire#powerrail
      Contact( "A07" )
   END_RUNG wire#w1
   RUNG wire#powerrail
      Contact( "A10" )
   END_RUNG wire#w1
   RUNG wire#powerrail
      Contact( "DB06_Clamp".dbx0_7 )
      Contact( "ConvOk3" )
   END_RUNG wire#w2
   // the same network as SCL:
   IF ((("M20.0" AND "DB03_Machine".dbx4_2) OR "A07" OR "A10") AND NOT "E72") OR ("DB06_Clamp".dbx0_7 AND "ConvOk3") THEN
       "DB23_AlarmProgram".dbx6_4 := TRUE;
   END_IF;
END_REGION

REGION Network 54: Alarm 54: Timeout for welder and cut unit forward/backward (Clam
   RUNG wire#powerrail
      Contact( "Timer".T82.Q )
      I_Contact( "Alarm" )
      S_Coil( "DB23_AlarmProgram".dbx6_5 )
   END_RUNG
   // the same network as SCL:
   IF "Timer".T82.Q AND NOT "Alarm" THEN "DB23_AlarmProgram".dbx6_5 := TRUE; END_IF;
END_REGION
END_FUNCTION

FUNCTION "FC18_ContrastCarriage" : Void   // FC18, LAD
TITLE = ContrastCarriage
{ S7_Optimized_Access := 'FALSE' }
VERSION : 0.1
// stored: AutoNumber false, IsIECCheckEnabled false, SetENOAutomatically false, UDAEnableTagReadback false
   VAR_TEMP   // added for the SCL form of the ladder/FBD networks
      _w1 : Bool;
   END_VAR
BEGIN

REGION Network 1: Timeout for welder contrast downward
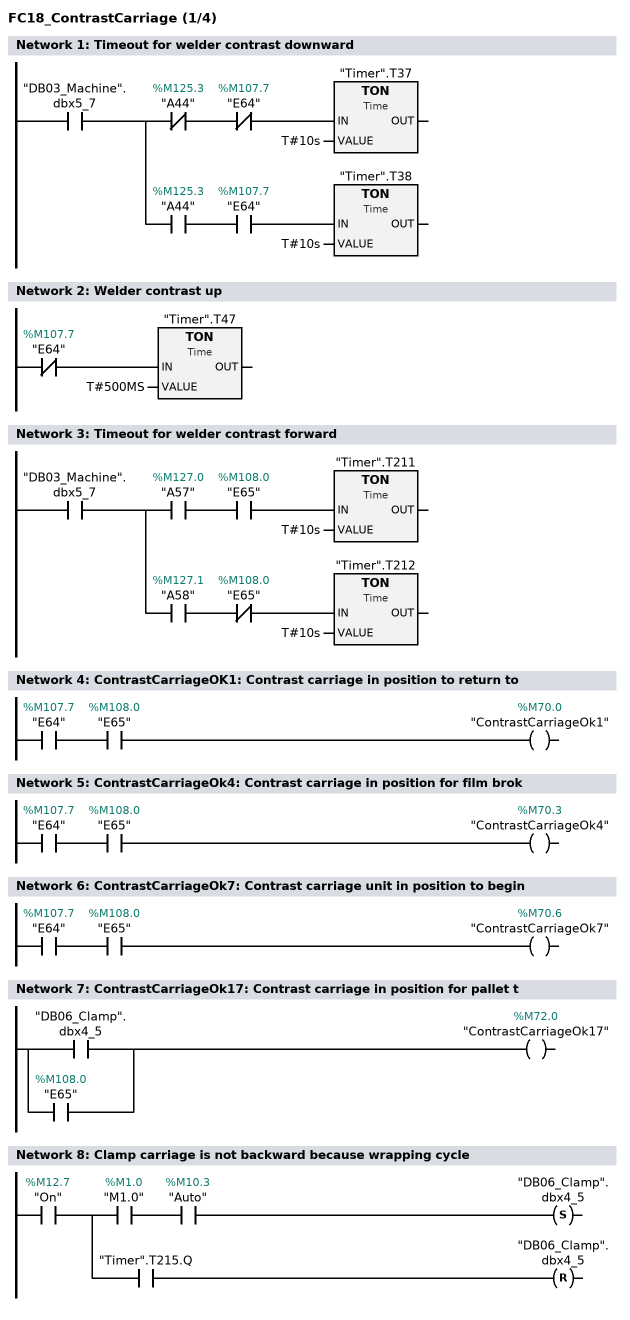
   "Timer".T37.TON(IN := "DB03_Machine".dbx5_7 AND NOT "A44" AND NOT "E64", PT := T#10s);   // TON coil
   "Timer".T38.TON(IN := "DB03_Machine".dbx5_7 AND "A44" AND "E64", PT := T#10s);   // TON coil
END_REGION

REGION Network 2: Welder contrast up
   "Timer".T47.TON(IN := NOT "E64", PT := T#500MS);   // TON coil
END_REGION

REGION Network 3: Timeout for welder contrast forward
   "Timer".T211.TON(IN := "DB03_Machine".dbx5_7 AND "A57" AND "E65", PT := T#10s);   // TON coil
   "Timer".T212.TON(IN := "DB03_Machine".dbx5_7 AND "A58" AND NOT "E65", PT := T#10s);   // TON coil
END_REGION

REGION Network 4: ContrastCarriageOK1: Contrast carriage in position to return to
   RUNG wire#powerrail
      Contact( "E64" )
      Contact( "E65" )
      Coil( "ContrastCarriageOk1" )
   END_RUNG
   // the same network as SCL:
   "ContrastCarriageOk1" := "E64" AND "E65";
END_REGION

REGION Network 5: ContrastCarriageOk4: Contrast carriage in position for film brok
   RUNG wire#powerrail
      Contact( "E64" )
      Contact( "E65" )
      Coil( "ContrastCarriageOk4" )
   END_RUNG
   // the same network as SCL:
   "ContrastCarriageOk4" := "E64" AND "E65";
END_REGION

REGION Network 6: ContrastCarriageOk7: Contrast carriage unit in position to begin
   RUNG wire#powerrail
      Contact( "E64" )
      Contact( "E65" )
      Coil( "ContrastCarriageOk7" )
   END_RUNG
   // the same network as SCL:
   "ContrastCarriageOk7" := "E64" AND "E65";
END_REGION

REGION Network 7: ContrastCarriageOk17: Contrast carriage in position for pallet t
   RUNG wire#powerrail
      Contact( "DB06_Clamp".dbx4_5 )
      wire#w1
      Coil( "ContrastCarriageOk17" )
   END_RUNG
   RUNG wire#powerrail
      Contact( "E65" )
   END_RUNG wire#w1
   // the same network as SCL:
   "ContrastCarriageOk17" := "DB06_Clamp".dbx4_5 OR "E65";
END_REGION

REGION Network 8: Clamp carriage is not backward because wrapping cycle
   RUNG wire#powerrail
      Contact( "On" )
      wire#w1
      Contact( "M1.0" )
      Contact( "Auto" )
      S_Coil( "DB06_Clamp".dbx4_5 )
   END_RUNG
   RUNG wire#w1
      Contact( "Timer".T215.Q )
      R_Coil( "DB06_Clamp".dbx4_5 )
   END_RUNG
   // the same network as SCL:
   IF "On" AND "M1.0" AND "Auto" THEN "DB06_Clamp".dbx4_5 := TRUE; END_IF;
   IF "On" AND "Timer".T215.Q THEN "DB06_Clamp".dbx4_5 := FALSE; END_IF;
END_REGION

REGION Network 9
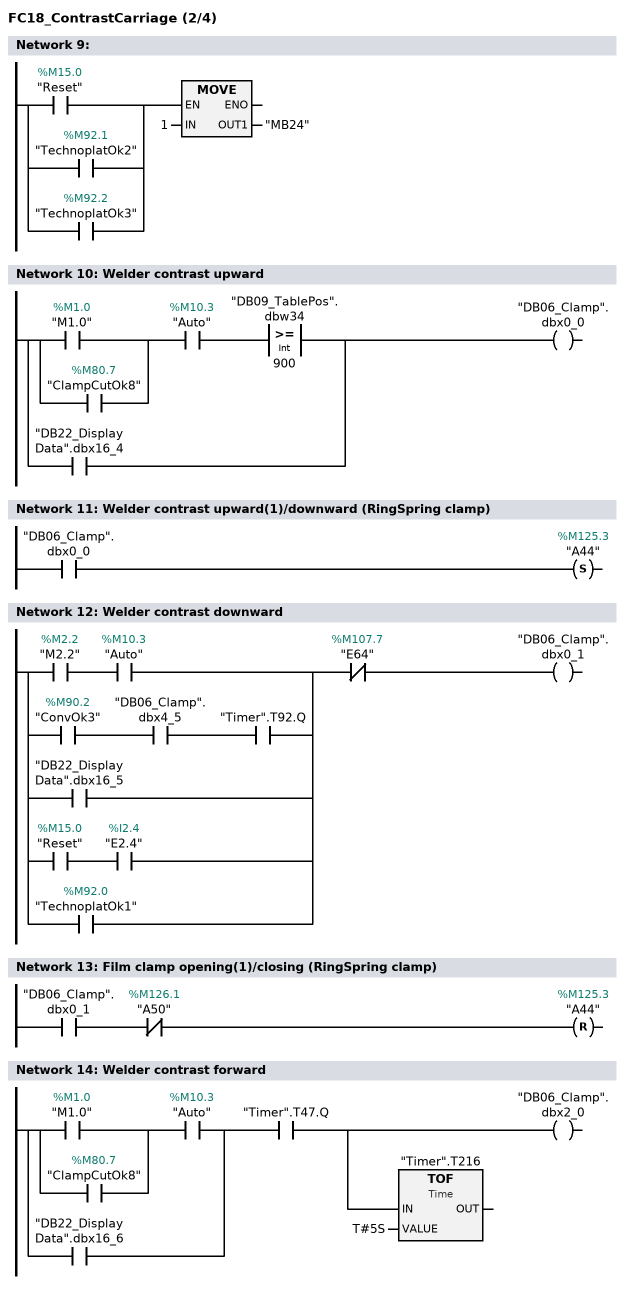
   RUNG wire#powerrail
      Contact( "Reset" )
      wire#w1
      { S7_GenerateENO := "TRUE" } Move(in := 1, out1 => "MB24")
   END_RUNG
   RUNG wire#powerrail
      Contact( "TechnoplatOk2" )
   END_RUNG wire#w1
   RUNG wire#powerrail
      Contact( "TechnoplatOk3" )
   END_RUNG wire#w1
   // the same network as SCL:
   IF "Reset" OR "TechnoplatOk2" OR "TechnoplatOk3" THEN "MB24" := 1; END_IF;
END_REGION

REGION Network 10: Welder contrast upward
   RUNG wire#powerrail
      Contact( "M1.0" )
      wire#w1
      Contact( "Auto" )
      { S7_Templates := "SrcType := Int" } GE_Contact(in1 := "DB09_TablePos".dbw34, in2 := 900)
      wire#w2
      Coil( "DB06_Clamp".dbx0_0 )
   END_RUNG
   RUNG wire#powerrail
      Contact( "ClampCutOk8" )
   END_RUNG wire#w1
   RUNG wire#powerrail
      Contact( "DB22_DisplayData".dbx16_4 )
   END_RUNG wire#w2
   // the same network as SCL:
   "DB06_Clamp".dbx0_0 := (("M1.0" OR "ClampCutOk8") AND "Auto" AND ("DB09_TablePos".dbw34 >= 900)) OR "DB22_DisplayData".dbx16_4;
END_REGION

REGION Network 11: Welder contrast upward(1)/downward (RingSpring clamp)
   RUNG wire#powerrail
      Contact( "DB06_Clamp".dbx0_0 )
      S_Coil( "A44" )
   END_RUNG
   // the same network as SCL:
   IF "DB06_Clamp".dbx0_0 THEN "A44" := TRUE; END_IF;
END_REGION

REGION Network 12: Welder contrast downward
   RUNG wire#powerrail
      Contact( "M2.2" )
      Contact( "Auto" )
      wire#w1
      I_Contact( "E64" )
      Coil( "DB06_Clamp".dbx0_1 )
   END_RUNG
   RUNG wire#powerrail
      Contact( "ConvOk3" )
      Contact( "DB06_Clamp".dbx4_5 )
      Contact( "Timer".T92.Q )
   END_RUNG wire#w1
   RUNG wire#powerrail
      Contact( "DB22_DisplayData".dbx16_5 )
   END_RUNG wire#w1
   RUNG wire#powerrail
      Contact( "Reset" )
      Contact( "E2.4" )
   END_RUNG wire#w1
   RUNG wire#powerrail
      Contact( "TechnoplatOk1" )
   END_RUNG wire#w1
   // the same network as SCL:
   "DB06_Clamp".dbx0_1 := (("M2.2" AND "Auto") OR ("ConvOk3" AND "DB06_Clamp".dbx4_5 AND "Timer".T92.Q) OR "DB22_DisplayData".dbx16_5 OR ("Reset" AND "E2.4") OR "TechnoplatOk1") AND NOT "E64";
END_REGION

REGION Network 13: Film clamp opening(1)/closing (RingSpring clamp)
   RUNG wire#powerrail
      Contact( "DB06_Clamp".dbx0_1 )
      I_Contact( "A50" )
      R_Coil( "A44" )
   END_RUNG
   // the same network as SCL:
   IF "DB06_Clamp".dbx0_1 AND NOT "A50" THEN "A44" := FALSE; END_IF;
END_REGION

REGION Network 14: Welder contrast forward
   "DB06_Clamp".dbx2_0 := ((("M1.0" OR "ClampCutOk8") AND "Auto") OR "DB22_DisplayData".dbx16_6) AND "Timer".T47.Q;
   "Timer".T216.TOF(IN := "DB06_Clamp".dbx2_0, PT := T#5S);   // TOF coil
END_REGION

REGION Network 15: Welder contrast forward(1)/backward (Contrast carriage)
